KUKA KRL program: MyProgram_330().src

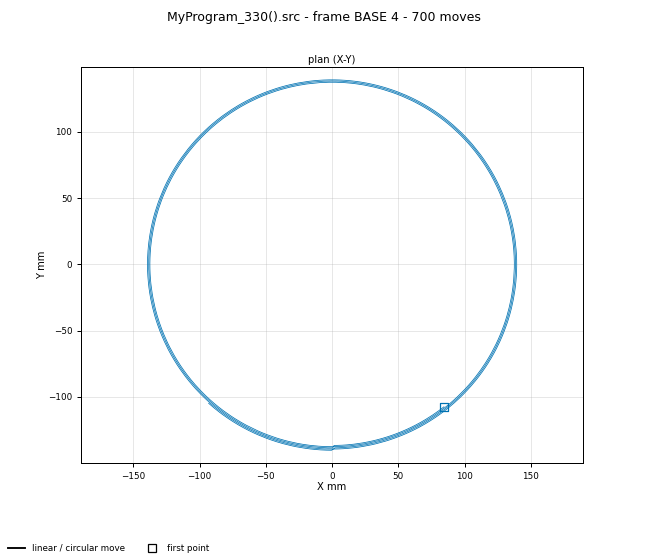
[picture p0: tool path of MyProgram_330().src in frame BASE 4, 700 of 700 moves have a stored position in this frame; points joined in program order, loops and branches not executed]
&ACCESS RVP
&REL 1
&PARAM TEMPLATE = C:\KRC\Roboter\Template\vorgabe
&PARAM EDITMASK = *
DEF MyProgram_330()
; ---- Setting reference (Base) ----
$BASE = BASE_DATA[4]

; --------------------------
; ---- Setting tool (TCP) ----
$TOOL = TOOL_DATA[3]
; --------------------------

$VEL.CP = VEL_APROX_PRINT
Startdeposition()
$VEL.CP = VEL_PRINT
LIN {X 84.385,Y -107.4322,Z 188,A -46.1092,B 2.2841,C 0.2483,E1 2.3985,E2 499.2761} C_DIS
LIN {X 80.7266,Y -110.2077,Z 188,A -48.0599,B 2.2837,C 0.2519,E1 2.3942,E2 501.2315} C_DIS
LIN {X 75.9214,Y -113.5713,Z 188,A -50.0705,B 2.2836,C 0.2529,E1 2.3897,E2 503.1841} C_DIS
LIN {X 73.4575,Y -115.1805,Z 188,A -51.7309,B 2.283,C 0.258,E1 2.3856,E2 504.9023} C_DIS
LIN {X 70.5993,Y -116.9539,Z 188,A -53.2982,B 2.2826,C 0.2614,E1 2.3818,E2 506.4914} C_DIS
LIN {X 66.6613,Y -119.2429,Z 188,A -54.7214,B 2.2826,C 0.2609,E1 2.3785,E2 507.8512} C_DIS
LIN {X 62.8545,Y -121.2922,Z 188,A -56.3872,B 2.2825,C 0.2626,E1 2.3744,E2 509.4986} C_DIS
LIN {X 59.8633,Y -122.7955,Z 188,A -57.8683,B 2.2822,C 0.2651,E1 2.3707,E2 510.991} C_DIS
LIN {X 56.2359,Y -124.4979,Z 188,A -59.8597,B 2.2817,C 0.2694,E1 2.3655,E2 513.0249} C_DIS
LIN {X 52.2998,Y -126.2016,Z 188,A -61.4901,B 2.2816,C 0.2705,E1 2.3614,E2 514.6342} C_DIS
LIN {X 48.8157,Y -127.5912,Z 188,A -62.7982,B 2.2816,C 0.2707,E1 2.358,E2 515.908} C_DIS
LIN {X 45.0187,Y -128.9782,Z 188,A -64.6024,B 2.2812,C 0.2733,E1 2.3532,E2 517.7279} C_DIS
LIN {X 41.9391,Y -130.0125,Z 188,A -65.4919,B 2.2814,C 0.2716,E1 2.351,E2 518.5549} C_DIS
LIN {X 37.8163,Y -131.2718,Z 188,A -67.5436,B 2.281,C 0.275,E1 2.3454,E2 520.6404} C_DIS
LIN {X 33.6424,Y -132.4016,Z 188,A -69.2051,B 2.281,C 0.2757,E1 2.341,E2 522.2827} C_DIS
LIN {X 30.2435,Y -133.2193,Z 188,A -70.6666,B 2.2808,C 0.2769,E1 2.337,E2 523.7444} C_DIS
LIN {X 26.7771,Y -133.9598,Z 188,A -72.0868,B 2.2808,C 0.2776,E1 2.3331,E2 525.1566} C_DIS
LIN {X 22.9551,Y -134.6675,Z 188,A -74.5642,B 2.2799,C 0.2839,E1 2.326,E2 527.7481} C_DIS
LIN {X 16.6479,Y -135.5918,Z 188,A -76.2129,B 2.2805,C 0.2793,E1 2.3218,E2 529.2614} C_DIS
LIN {X 10.9508,Y -136.1704,Z 188,A -78.8787,B 2.2802,C 0.282,E1 2.3143,E2 531.9641} C_DIS
LIN {X 7.4758,Y -136.4059,Z 188,A -80.9653,B 2.2797,C 0.2861,E1 2.3082,E2 534.1351} C_DIS
LIN {X 1.4605,Y -136.6033,Z 188,A -82.7052,B 2.2801,C 0.2824,E1 2.3036,E2 535.7715} C_DIS
LIN {X 1.4605,Y -136.6033,Z 188,A -82.7052,B 2.2801,C 0.2824,E1 2.3036,E2 535.7715} C_DIS
Enddeposition()
LIN {X 1.0092,Y -137.5035,Z 188,A -82.2384,B 2.2498,C 0.2786,E1 2.2744,E2 535.2539} C_DIS
Startdeposition()
$VEL.CP = VEL_PRINT
LIN {X 4.8877,Y -137.4225,Z 188,A -80.4582,B 2.25,C 0.2772,E1 2.2795,E2 533.4505} C_DIS
LIN {X 9.447,Y -137.1848,Z 188,A -78.1611,B 2.2504,C 0.2742,E1 2.2861,E2 531.0981} C_DIS
LIN {X 14.028,Y -136.7928,Z 188,A -76.6474,B 2.2502,C 0.2756,E1 2.2901,E2 529.6387} C_DIS
LIN {X 20.7914,Y -135.9277,Z 188,A -73.7592,B 2.2504,C 0.2736,E1 2.2982,E2 526.7425} C_DIS
LIN {X 24.9857,Y -135.2215,Z 188,A -71.9483,B 2.2506,C 0.2722,E1 2.3032,E2 524.9253} C_DIS
LIN {X 28.2124,Y -134.5853,Z 188,A -70.7396,B 2.2506,C 0.2722,E1 2.3064,E2 523.738} C_DIS
LIN {X 32.1471,Y -133.6978,Z 188,A -69.2265,B 2.2506,C 0.2718,E1 2.3105,E2 522.2468} C_DIS
LIN {X 35.1427,Y -132.9421,Z 188,A -67.9438,B 2.2508,C 0.2706,E1 2.3139,E2 520.9639} C_DIS
LIN {X 38.5637,Y -131.99,Z 188,A -66.5352,B 2.2508,C 0.2697,E1 2.3177,E2 519.564} C_DIS
LIN {X 41.3681,Y -131.139,Z 188,A -65.2923,B 2.2511,C 0.2683,E1 2.321,E2 518.3174} C_DIS
LIN {X 44.7036,Y -130.0393,Z 188,A -64.0619,B 2.2511,C 0.2683,E1 2.3242,E2 517.1178} C_DIS
LIN {X 47.8191,Y -128.9264,Z 188,A -62.5742,B 2.2513,C 0.2659,E1 2.3282,E2 515.6143} C_DIS
LIN {X 54.9877,Y -126.0358,Z 188,A -59.4365,B 2.2517,C 0.2625,E1 2.3363,E2 512.4858} C_DIS
LIN {X 58.7508,Y -124.3268,Z 188,A -57.6919,B 2.252,C 0.26,E1 2.3407,E2 510.737} C_DIS
LIN {X 62.1581,Y -122.6576,Z 188,A -56.2754,B 2.2522,C 0.2589,E1 2.3442,E2 509.3417} C_DIS
LIN {X 64.9016,Y -121.2305,Z 188,A -54.4156,B 2.2528,C 0.253,E1 2.349,E2 507.403} C_DIS
LIN {X 69.1543,Y -118.8562,Z 188,A -52.9164,B 2.2528,C 0.2536,E1 2.3525,E2 505.9749} C_DIS
LIN {X 72.9516,Y -116.5642,Z 188,A -51.1222,B 2.2531,C 0.251,E1 2.3567,E2 504.1867} C_DIS
LIN {X 77.4592,Y -113.6185,Z 188,A -48.9633,B 2.2534,C 0.2478,E1 2.3617,E2 502.0377} C_DIS
LIN {X 81.2164,Y -110.9639,Z 188,A -47.1203,B 2.2537,C 0.2449,E1 2.3659,E2 500.2032} C_DIS
LIN {X 84.798,Y -108.2513,Z 188,A -45.3204,B 2.254,C 0.242,E1 2.3699,E2 498.4117} C_DIS
LIN {X 88.2179,Y -105.483,Z 188,A -43.5989,B 2.2543,C 0.2394,E1 2.3735,E2 496.7039} C_DIS
LIN {X 91.488,Y -102.66,Z 188,A -41.8357,B 2.2547,C 0.2361,E1 2.3772,E2 494.9444} C_DIS
LIN {X 94.8941,Y -99.5196,Z 188,A -39.9954,B 2.255,C 0.2329,E1 2.381,E2 493.1147} C_DIS
LIN {X 98.0963,Y -96.3647,Z 188,A -38.3712,B 2.2552,C 0.2308,E1 2.3841,E2 491.5226} C_DIS
LIN {X 100.1859,Y -94.1905,Z 188,A -36.9746,B 2.2556,C 0.2271,E1 2.3868,E2 490.1062} C_DIS
LIN {X 103.1659,Y -90.9168,Z 188,A -35.2946,B 2.2559,C 0.2243,E1 2.3899,E2 488.447} C_DIS
LIN {X 105.9358,Y -87.6734,Z 188,A -33.5608,B 2.2562,C 0.2207,E1 2.393,E2 486.7176} C_DIS
LIN {X 108.3988,Y -84.6101,Z 188,A -31.9453,B 2.2566,C 0.2171,E1 2.3958,E2 485.1038} C_DIS
LIN {X 112.2568,Y -79.4196,Z 188,A -28.7306,B 2.2575,C 0.2067,E1 2.4012,E2 481.8167} C_DIS
LIN {X 115.783,Y -74.1843,Z 188,A -26.5211,B 2.2578,C 0.2037,E1 2.4045,E2 479.6621} C_DIS
LIN {X 118.237,Y -70.2074,Z 188,A -25.0755,B 2.2578,C 0.2029,E1 2.4064,E2 478.2823} C_DIS
LIN {X 120.3276,Y -66.5604,Z 188,A -23.5052,B 2.2582,C 0.2,E1 2.4086,E2 476.7348} C_DIS
LIN {X 122.3374,Y -62.7871,Z 188,A -21.8144,B 2.2585,C 0.1962,E1 2.4107,E2 475.0547} C_DIS
LIN {X 123.689,Y -60.0848,Z 188,A -20.6209,B 2.2587,C 0.1935,E1 2.4122,E2 473.869} C_DIS
LIN {X 125.4096,Y -56.4002,Z 188,A -19.1302,B 2.2589,C 0.1908,E1 2.4139,E2 472.404} C_DIS
LIN {X 127.1795,Y -52.2917,Z 188,A -17.2805,B 2.2593,C 0.186,E1 2.4159,E2 470.5549} C_DIS
LIN {X 128.6189,Y -48.64,Z 188,A -15.725,B 2.2596,C 0.1823,E1 2.4175,E2 469.0087} C_DIS
LIN {X 129.6006,Y -45.964,Z 188,A -14.34,B 2.26,C 0.1775,E1 2.4188,E2 467.5967} C_DIS
LIN {X 130.667,Y -42.8375,Z 188,A -13.3208,B 2.26,C 0.1768,E1 2.4197,E2 466.6238} C_DIS
LIN {X 131.8901,Y -38.905,Z 188,A -11.6877,B 2.2604,C 0.1728,E1 2.421,E2 465.0003} C_DIS
LIN {X 132.827,Y -35.5744,Z 188,A -10.3764,B 2.2606,C 0.17,E1 2.4219,E2 463.7052} C_DIS
LIN {X 133.5449,Y -32.7814,Z 188,A -9.1356,B 2.2609,C 0.1663,E1 2.4228,E2 462.4583} C_DIS
LIN {X 134.3884,Y -29.1259,Z 188,A -7.7687,B 2.2611,C 0.1637,E1 2.4236,E2 461.1161} C_DIS
LIN {X 135.0373,Y -25.9515,Z 188,A -6.4806,B 2.2613,C 0.1604,E1 2.4243,E2 459.8352} C_DIS
LIN {X 135.6371,Y -22.6082,Z 188,A -4.5754,B 2.2619,C 0.1524,E1 2.4252,E2 457.8646} C_DIS
LIN {X 136.364,Y -17.7048,Z 188,A -3.254,B 2.2619,C 0.1529,E1 2.4257,E2 456.6394} C_DIS
LIN {X 137.0505,Y -11.2195,Z 188,A -0.508,B 2.2623,C 0.145,E1 2.4264,E2 453.8881} C_DIS
LIN {X 137.4867,Y -2.4643,Z 188,A 3.1629,B 2.263,C 0.1346,E1 2.4268,E2 450.2126} C_DIS
LIN {X 137.5031,Y 1.4155,Z 188,A 4.4461,B 2.263,C 0.1328,E1 2.4268,E2 448.9718} C_DIS
LIN {X 137.3718,Y 6.1756,Z 188,A 6.7563,B 2.2636,C 0.1246,E1 2.4265,E2 446.6181} C_DIS
LIN {X 137.064,Y 11.0604,Z 188,A 8.1298,B 2.2636,C 0.1243,E1 2.4262,E2 445.3298} C_DIS
LIN {X 136.5849,Y 15.9147,Z 188,A 10.3416,B 2.264,C 0.1172,E1 2.4256,E2 443.0936} C_DIS
LIN {X 136.139,Y 19.3583,Z 188,A 11.2132,B 2.264,C 0.1179,E1 2.4253,E2 442.2952} C_DIS
LIN {X 135.4537,Y 23.6884,Z 188,A 13.1868,B 2.2642,C 0.1116,E1 2.4244,E2 440.3019} C_DIS
LIN {X 134.7483,Y 27.4126,Z 188,A 14.6147,B 2.2644,C 0.1085,E1 2.4236,E2 438.8925} C_DIS
LIN {X 133.981,Y 30.9474,Z 188,A 16.1028,B 2.2646,C 0.1045,E1 2.4227,E2 437.4062} C_DIS
LIN {X 132.9463,Y 35.1268,Z 188,A 17.7419,B 2.2647,C 0.1008,E1 2.4216,E2 435.786} C_DIS
LIN {X 132.0775,Y 38.2649,Z 188,A 18.8829,B 2.2648,C 0.0989,E1 2.4207,E2 434.6718} C_DIS
LIN {X 131.1193,Y 41.4299,Z 188,A 20.3392,B 2.265,C 0.0945,E1 2.4195,E2 433.2049} C_DIS
LIN {X 130.0245,Y 44.7462,Z 188,A 21.7058,B 2.2651,C 0.0913,E1 2.4183,E2 431.8489} C_DIS
LIN {X 126.6388,Y 53.5863,Z 188,A 25.2973,B 2.2654,C 0.0838,E1 2.4147,E2 428.3006} C_DIS
LIN {X 124.7724,Y 57.7956,Z 188,A 27.17,B 2.2656,C 0.0792,E1 2.4126,E2 426.4331} C_DIS
LIN {X 123.3269,Y 60.8189,Z 188,A 28.5186,B 2.2657,C 0.076,E1 2.4109,E2 425.09} C_DIS
LIN {X 121.8441,Y 63.7378,Z 188,A 29.7762,B 2.2657,C 0.0733,E1 2.4093,E2 423.8453} C_DIS
LIN {X 119.9629,Y 67.2158,Z 188,A 31.2497,B 2.2659,C 0.0706,E1 2.4074,E2 422.3931} C_DIS
LIN {X 118.3323,Y 70.0475,Z 188,A 32.7955,B 2.266,C 0.0658,E1 2.4051,E2 420.8239} C_DIS
LIN {X 115.9995,Y 73.8462,Z 188,A 34.3445,B 2.266,C 0.0636,E1 2.4029,E2 419.313} C_DIS
LIN {X 113.911,Y 77.028,Z 188,A 36.0298,B 2.2662,C 0.0591,E1 2.4003,E2 417.6148} C_DIS
LIN {X 111.2107,Y 80.878,Z 188,A 37.8786,B 2.2663,C 0.0553,E1 2.3973,E2 415.7793} C_DIS
LIN {X 108.5058,Y 84.4725,Z 188,A 39.6601,B 2.2663,C 0.0517,E1 2.3943,E2 414.0091} C_DIS
LIN {X 105.801,Y 87.8362,Z 188,A 41.375,B 2.2665,C 0.0483,E1 2.3913,E2 412.3041} C_DIS
LIN {X 102.8084,Y 91.3211,Z 188,A 43.0061,B 2.2665,C 0.0462,E1 2.3884,E2 410.7077} C_DIS
LIN {X 100.499,Y 93.8563,Z 188,A 44.5615,B 2.2665,C 0.0422,E1 2.3854,E2 409.1366} C_DIS
LIN {X 97.3828,Y 97.0858,Z 188,A 46.258,B 2.2666,C 0.0396,E1 2.3821,E2 407.4612} C_DIS
LIN {X 94.6427,Y 99.7593,Z 188,A 47.9247,B 2.2667,C 0.0358,E1 2.3787,E2 405.7856} C_DIS
LIN {X 90.7645,Y 103.3005,Z 188,A 49.998,B 2.2667,C 0.0323,E1 2.3744,E2 403.7263} C_DIS
LIN {X 87.3118,Y 106.2347,Z 188,A 51.8087,B 2.2667,C 0.0293,E1 2.3706,E2 401.9249} C_DIS
LIN {X 83.8262,Y 109.0061,Z 188,A 53.61,B 2.2668,C 0.0262,E1 2.3666,E2 400.1302} C_DIS
LIN {X 80.1135,Y 111.7625,Z 188,A 55.4244,B 2.2668,C 0.0236,E1 2.3625,E2 398.3296} C_DIS
LIN {X 76.6335,Y 114.1772,Z 188,A 56.9231,B 2.2668,C 0.0224,E1 2.3592,E2 396.8635} C_DIS
LIN {X 73.842,Y 116.0022,Z 188,A 58.4469,B 2.2669,C 0.0192,E1 2.3555,E2 395.3233} C_DIS
LIN {X 70.038,Y 118.338,Z 188,A 60.482,B 2.2669,C 0.0151,E1 2.3506,E2 393.267} C_DIS
LIN {X 67.0583,Y 120.0514,Z 188,A 61.6697,B 2.2669,C 0.0146,E1 2.3478,E2 392.1093} C_DIS
LIN {X 62.7474,Y 122.3576,Z 188,A 63.5951,B 2.2669,C 0.0123,E1 2.343,E2 390.1975} C_DIS
LIN {X 59.8978,Y 123.7788,Z 188,A 65.8423,B 2.2669,C 0.0047,E1 2.3371,E2 387.8377} C_DIS
LIN {X 53.1857,Y 126.8061,Z 188,A 67.5662,B 2.2669,C 0.0092,E1 2.3331,E2 386.2787} C_DIS
LIN {X 49.184,Y 128.4129,Z 188,A 69.6653,B 2.2669,C 0.0052,E1 2.3275,E2 384.1434} C_DIS
LIN {X 45.5722,Y 129.7381,Z 188,A 71.2409,B 2.2669,C 0.0036,E1 2.3234,E2 382.5715} C_DIS
LIN {X 41.6932,Y 131.0351,Z 188,A 72.7706,B 2.2669,C 0.0029,E1 2.3194,E2 381.0632} C_DIS
LIN {X 38.8098,Y 131.918,Z 188,A 73.9119,B 2.2669,C 0.0024,E1 2.3163,E2 379.9361} C_DIS
LIN {X 35.34,Y 132.8895,Z 188,A 75.5057,B 2.2669,C 0.0005,E1 2.312,E2 378.3315} C_DIS
LIN {X 31.2031,Y 133.9226,Z 188,A 77.3013,B 2.2669,C -0.0011,E1 2.3071,E2 376.5341} C_DIS
LIN {X 26.966,Y 134.8391,Z 188,A 79.1348,B 2.2669,C -0.0026,E1 2.3021,E2 374.6979} C_DIS
LIN {X 24,Y 135.3979,Z 188,A 80.9141,B 2.2669,C -0.0063,E1 2.297,E2 372.8556} C_DIS
LIN {X 18.5994,Y 136.2463,Z 188,A 82.5017,B 2.2669,C -0.0038,E1 2.2929,E2 371.3526} C_DIS
LIN {X 14.7664,Y 136.7133,Z 188,A 84.1663,B 2.2669,C -0.0049,E1 2.2882,E2 369.6818} C_DIS
LIN {X 9.7967,Y 137.1593,Z 188,A 86.1603,B 2.2669,C -0.0053,E1 2.2827,E2 367.6988} C_DIS
LIN {X 5.5957,Y 137.3949,Z 188,A 87.923,B 2.2669,C -0.0059,E1 2.2777,E2 365.9356} C_DIS
LIN {X 2.7166,Y 137.4825,Z 188,A 89.6743,B 2.2669,C -0.009,E1 2.2727,E2 364.1183} C_DIS
LIN {X -2.2082,Y 137.4909,Z 188,A 91.1797,B 2.2669,C -0.0066,E1 2.2686,E2 362.6798} C_DIS
LIN {X -9.3667,Y 137.1907,Z 188,A 94.2648,B 2.2669,C -0.0072,E1 2.26,E2 359.5841} C_DIS
LIN {X -19.2271,Y 136.1578,Z 188,A 98.2457,B 2.2669,C -0.0059,E1 2.249,E2 355.6234} C_DIS
LIN {X -22.1843,Y 135.7078,Z 188,A 99.3663,B 2.2669,C -0.005,E1 2.2459,E2 354.5186} C_DIS
LIN {X -25.6321,Y 135.0984,Z 188,A 100.9338,B 2.2669,C -0.005,E1 2.2416,E2 352.9388} C_DIS
LIN {X -28.9391,Y 134.4287,Z 188,A 102.2586,B 2.2669,C -0.0041,E1 2.2379,E2 351.6244} C_DIS
LIN {X -31.8422,Y 133.7713,Z 188,A 103.5303,B 2.2669,C -0.0037,E1 2.2345,E2 350.3497} C_DIS
LIN {X -35.1431,Y 132.942,Z 188,A 105.0418,B 2.2669,C -0.0033,E1 2.2303,E2 348.8277} C_DIS
LIN {X -37.9505,Y 132.1695,Z 188,A 106.3797,B 2.2669,C -0.0031,E1 2.2267,E2 347.4755} C_DIS
LIN {X -42.3548,Y 130.8238,Z 188,A 109.2577,B 2.2669,C -0.0056,E1 2.2188,E2 344.4824} C_DIS
LIN {X -49.02,Y 128.4766,Z 188,A 111.4022,B 2.2669,C -0.0001,E1 2.2134,E2 342.4369} C_DIS
LIN {X -51.732,Y 127.4064,Z 188,A 112.9877,B 2.2669,C -0.0004,E1 2.2092,E2 340.8072} C_DIS
LIN {X -55.7214,Y 125.7132,Z 188,A 114.397,B 2.2669,C 0.0028,E1 2.2057,E2 339.4471} C_DIS
LIN {X -59.0649,Y 124.1767,Z 188,A 115.8846,B 2.2669,C 0.0046,E1 2.2019,E2 337.9659} C_DIS
LIN {X -61.9449,Y 122.7661,Z 188,A 117.3342,B 2.2669,C 0.0056,E1 2.1982,E2 336.5036} C_DIS
LIN {X -64.7223,Y 121.3269,Z 188,A 118.7822,B 2.2669,C 0.0067,E1 2.1946,E2 335.039} C_DIS
LIN {X -68.9997,Y 118.9457,Z 188,A 120.7472,B 2.2669,C 0.0095,E1 2.1899,E2 333.0843} C_DIS
LIN {X -72.4713,Y 116.863,Z 188,A 122.6066,B 2.2669,C 0.0111,E1 2.1854,E2 331.2051} C_DIS
LIN {X -76.5464,Y 114.2354,Z 188,A 124.6275,B 2.2669,C 0.014,E1 2.1807,E2 329.1856} C_DIS
LIN {X -82.1038,Y 110.3086,Z 188,A 128.5193,B 2.2669,C 0.0151,E1 2.1716,E2 325.1665} C_DIS
LIN {X -87.6822,Y 105.9285,Z 188,A 131.1917,B 2.2669,C 0.0209,E1 2.1659,E2 322.531} C_DIS
LIN {X -91.5102,Y 102.64,Z 188,A 133.0073,B 2.2669,C 0.0254,E1 2.1622,E2 320.7521} C_DIS
LIN {X -95.4132,Y 99.0224,Z 188,A 135.1786,B 2.2668,C 0.0296,E1 2.1578,E2 318.5881} C_DIS
LIN {X -98.6463,Y 95.8017,Z 188,A 137.8599,B 2.2668,C 0.0311,E1 2.1524,E2 315.8122} C_DIS
LIN {X -102.6929,Y 91.4512,Z 188,A 139.5412,B 2.2667,C 0.0382,E1 2.1494,E2 314.2306} C_DIS
LIN {X -104.73,Y 89.1103,Z 188,A 141.5886,B 2.2667,C 0.0389,E1 2.1455,E2 312.0913} C_DIS
LIN {X -107.7808,Y 85.3956,Z 188,A 143.0983,B 2.2665,C 0.0444,E1 2.143,E2 310.6439} C_DIS
LIN {X -110.484,Y 81.8683,Z 188,A 145.1289,B 2.2665,C 0.048,E1 2.1395,E2 308.5927} C_DIS
LIN {X -112.9783,Y 78.3897,Z 188,A 146.9931,B 2.2664,C 0.0518,E1 2.1365,E2 306.7198} C_DIS
LIN {X -115.3932,Y 74.7893,Z 188,A 148.9146,B 2.2664,C 0.0557,E1 2.1335,E2 304.7854} C_DIS
LIN {X -117.1838,Y 71.9513,Z 188,A 150.7097,B 2.2662,C 0.0581,E1 2.1309,E2 302.9422} C_DIS
LIN {X -119.1363,Y 68.6704,Z 188,A 152.0071,B 2.2662,C 0.0625,E1 2.1291,E2 301.6824} C_DIS
LIN {X -121.3269,Y 64.7222,Z 188,A 154.1462,B 2.266,C 0.0665,E1 2.1262,E2 299.5126} C_DIS
LIN {X -123.331,Y 60.8105,Z 188,A 155.8989,B 2.2659,C 0.0712,E1 2.124,E2 297.771} C_DIS
LIN {X -124.5803,Y 58.211,Z 188,A 157.261,B 2.2658,C 0.0739,E1 2.1224,E2 296.3898} C_DIS
LIN {X -125.9787,Y 55.1199,Z 188,A 158.7316,B 2.2657,C 0.0774,E1 2.1207,E2 294.9131} C_DIS
LIN {X -127.2677,Y 52.0761,Z 188,A 160.275,B 2.2656,C 0.0806,E1 2.119,E2 293.35} C_DIS
LIN {X -128.6839,Y 48.4665,Z 188,A 161.8237,B 2.2654,C 0.0849,E1 2.1175,E2 291.8108} C_DIS
LIN {X -129.8655,Y 45.2048,Z 188,A 163.2663,B 2.2652,C 0.0887,E1 2.1161,E2 290.3696} C_DIS
LIN {X -130.721,Y 42.6749,Z 188,A 164.6068,B 2.2652,C 0.0912,E1 2.1149,E2 289.0014} C_DIS
LIN {X -131.9233,Y 38.7915,Z 188,A 166.4002,B 2.265,C 0.0955,E1 2.1135,E2 287.1967} C_DIS
LIN {X -133.2108,Y 34.1098,Z 188,A 168.5508,B 2.2647,C 0.1008,E1 2.1119,E2 285.0314} C_DIS
LIN {X -134.0307,Y 30.7299,Z 188,A 170.202,B 2.2646,C 0.1043,E1 2.1108,E2 283.3558} C_DIS
LIN {X -135.0028,Y 26.1323,Z 188,A 172.2053,B 2.2643,C 0.1096,E1 2.1097,E2 281.348} C_DIS
LIN {X -135.6278,Y 22.6641,Z 188,A 173.719,B 2.2641,C 0.1136,E1 2.109,E2 279.8296} C_DIS
LIN {X -136.0754,Y 19.8037,Z 188,A 175.0268,B 2.264,C 0.1167,E1 2.1084,E2 278.5098} C_DIS
LIN {X -136.4612,Y 16.9522,Z 188,A 176.4374,B 2.2638,C 0.1197,E1 2.1079,E2 277.073} C_DIS
LIN {X -136.9105,Y 12.8145,Z 188,A 178.2497,B 2.2636,C 0.1244,E1 2.1074,E2 275.252} C_DIS
LIN {X -137.2408,Y 8.5783,Z 188,A -179.9451,B 2.2633,C 0.1293,E1 2.1071,E2 273.4434} C_DIS
LIN {X -137.428,Y 4.7461,Z 188,A -178.274,B 2.263,C 0.1336,E1 2.1069,E2 271.7641} C_DIS
LIN {X -137.5082,Y 0.6532,Z 188,A -176.3294,B 2.2628,C 0.138,E1 2.1068,E2 269.7899} C_DIS
LIN {X -137.4625,Y -3.5713,Z 188,A -174.5103,B 2.2625,C 0.1428,E1 2.1068,E2 267.9644} C_DIS
LIN {X -137.3184,Y -7.2363,Z 188,A -172.8003,B 2.2622,C 0.1467,E1 2.1071,E2 266.2318} C_DIS
LIN {X -137.0681,Y -11.0116,Z 188,A -171.1578,B 2.262,C 0.151,E1 2.1075,E2 264.5817} C_DIS
LIN {X -136.6969,Y -14.9194,Z 188,A -169.4434,B 2.2617,C 0.1554,E1 2.108,E2 262.8581} C_DIS
LIN {X -136.1792,Y -19.0769,Z 188,A -167.5781,B 2.2613,C 0.16,E1 2.1086,E2 260.9783} C_DIS
LIN {X -135.7078,Y -22.1843,Z 188,A -166.274,B 2.2611,C 0.1636,E1 2.1092,E2 259.6756} C_DIS
LIN {X -135.1272,Y -25.4818,Z 188,A -164.6905,B 2.2608,C 0.1671,E1 2.11,E2 258.0683} C_DIS
LIN {X -134.4414,Y -28.8803,Z 188,A -163.2603,B 2.2605,C 0.1711,E1 2.1108,E2 256.6408} C_DIS
LIN {X -133.7519,Y -31.9227,Z 188,A -161.8533,B 2.2603,C 0.1744,E1 2.1117,E2 255.2205} C_DIS
LIN {X -133.0511,Y -34.7339,Z 188,A -160.4123,B 2.2601,C 0.1771,E1 2.1128,E2 253.7496} C_DIS
LIN {X -132.0466,Y -38.3704,Z 188,A -158.8371,B 2.2597,C 0.1813,E1 2.114,E2 252.1747} C_DIS
LIN {X -130.2796,Y -44.0009,Z 188,A -156.1023,B 2.2592,C 0.1872,E1 2.1163,E2 249.4049} C_DIS
LIN {X -128.555,Y -48.8107,Z 188,A -153.8695,B 2.2588,C 0.1925,E1 2.1185,E2 247.1593} C_DIS
LIN {X -126.9886,Y -52.7487,Z 188,A -152.0935,B 2.2584,C 0.197,E1 2.1204,E2 245.3827} C_DIS
LIN {X -125.5772,Y -56.0254,Z 188,A -150.6125,B 2.2581,C 0.2008,E1 2.122,E2 243.903} C_DIS
LIN {X -124.1951,Y -59.0265,Z 188,A -149.0837,B 2.2578,C 0.2039,E1 2.1239,E2 242.3546} C_DIS
LIN {X -122.6701,Y -62.1335,Z 188,A -147.5877,B 2.2575,C 0.2073,E1 2.1257,E2 240.8521} C_DIS
LIN {X -119.0182,Y -68.8745,Z 188,A -144.0569,B 2.2569,C 0.2141,E1 2.1306,E2 237.2779} C_DIS
LIN {X -116.6028,Y -72.8896,Z 188,A -141.9949,B 2.2564,C 0.2184,E1 2.1336,E2 235.2019} C_DIS
LIN {X -114.1602,Y -76.6591,Z 188,A -140.0279,B 2.2561,C 0.2223,E1 2.1366,E2 233.2228} C_DIS
LIN {X -111.6162,Y -80.3182,Z 188,A -138.0713,B 2.2557,C 0.2262,E1 2.1398,E2 231.2532} C_DIS
LIN {X -108.9478,Y -83.9022,Z 188,A -136.1116,B 2.2553,C 0.2299,E1 2.1431,E2 229.2809} C_DIS
LIN {X -106.2091,Y -87.3431,Z 188,A -134.1535,B 2.255,C 0.2333,E1 2.1466,E2 227.3063} C_DIS
LIN {X -103.5532,Y -90.4752,Z 188,A -131.6718,B 2.2548,C 0.2344,E1 2.1514,E2 224.7208} C_DIS
LIN {X -99.5157,Y -94.8982,Z 188,A -129.96,B 2.2541,C 0.2417,E1 2.1544,E2 223.1153} C_DIS
LIN {X -95.4652,Y -98.9721,Z 188,A -127.3581,B 2.2537,C 0.2455,E1 2.1597,E2 220.4857} C_DIS
LIN {X -92.369,Y -101.8675,Z 188,A -125.4795,B 2.2534,C 0.2482,E1 2.1636,E2 218.5922} C_DIS
LIN {X -88.9812,Y -104.8397,Z 188,A -123.4974,B 2.253,C 0.2511,E1 2.1678,E2 216.596} C_DIS
LIN {X -85.4608,Y -107.7289,Z 188,A -121.5416,B 2.2527,C 0.2539,E1 2.1721,E2 214.6324} C_DIS
LIN {X -81.8426,Y -110.5031,Z 188,A -119.549,B 2.2524,C 0.2565,E1 2.1765,E2 212.6273} C_DIS
LIN {X -79.3508,Y -112.3053,Z 188,A -118.042,B 2.2524,C 0.2576,E1 2.1801,E2 211.0896} C_DIS
LIN {X -76.6488,Y -114.167,Z 188,A -116.7829,B 2.252,C 0.2599,E1 2.1829,E2 209.8452} C_DIS
LIN {X -73.3109,Y -116.338,Z 188,A -114.9317,B 2.2519,C 0.2614,E1 2.1874,E2 207.9677} C_DIS
LIN {X -68.5317,Y -119.2166,Z 188,A -112.7023,B 2.2515,C 0.2647,E1 2.1927,E2 205.7512} C_DIS
LIN {X -64.629,Y -121.3762,Z 188,A -110.7882,B 2.2513,C 0.2666,E1 2.1974,E2 203.8293} C_DIS
LIN {X -56.1373,Y -125.5272,Z 188,A -107.0196,B 2.2507,C 0.2714,E1 2.2069,E2 200.0833} C_DIS
LIN {X -52.6904,Y -127.013,Z 188,A -105.2755,B 2.2507,C 0.272,E1 2.2114,E2 198.3144} C_DIS
LIN {X -48.9416,Y -128.5059,Z 188,A -103.3797,B 2.2506,C 0.2724,E1 2.2165,E2 196.3891} C_DIS
LIN {X -45.0592,Y -129.916,Z 188,A -101.8833,B 2.2503,C 0.2747,E1 2.2203,E2 194.9229} C_DIS
LIN {X -42.0191,Y -130.931,Z 188,A -100.5596,B 2.2502,C 0.2757,E1 2.2238,E2 193.6005} C_DIS
LIN {X -39.4366,Y -131.7344,Z 188,A -99.1642,B 2.2502,C 0.2751,E1 2.2277,E2 192.1682} C_DIS
LIN {X -35.8085,Y -132.7645,Z 188,A -97.6957,B 2.2501,C 0.2765,E1 2.2316,E2 190.7132} C_DIS
LIN {X -32.4912,Y -133.6149,Z 188,A -96.2887,B 2.25,C 0.2772,E1 2.2354,E2 189.3085} C_DIS
LIN {X -29.1508,Y -134.383,Z 188,A -94.8386,B 2.25,C 0.2777,E1 2.2394,E2 187.8549} C_DIS
LIN {X -26.43,Y -134.9459,Z 188,A -93.2028,B 2.2502,C 0.2757,E1 2.2441,E2 186.1531} C_DIS
LIN {X -22.2736,Y -135.6929,Z 188,A -91.9109,B 2.2498,C 0.2785,E1 2.2475,E2 184.9248} C_DIS
LIN {X -17.0251,Y -136.4523,Z 188,A -89.5947,B 2.2498,C 0.2783,E1 2.2539,E2 182.5932} C_DIS
LIN {X -13.3974,Y -136.8545,Z 188,A -88.2108,B 2.2498,C 0.2792,E1 2.2577,E2 181.2274} C_DIS
LIN {X -10.1008,Y -137.1371,Z 188,A -86.7431,B 2.2498,C 0.2787,E1 2.2619,E2 179.7468} C_DIS
LIN {X -5.8583,Y -137.3847,Z 188,A -85.1488,B 2.2497,C 0.2795,E1 2.2663,E2 178.176} C_DIS
LIN {X -2.4585,Y -137.4868,Z 188,A -83.3294,B 2.25,C 0.2771,E1 2.2715,E2 176.3007} C_DIS
LIN {X 1.0092,Y -137.5035,Z 188,A -82.2352,B 2.2498,C 0.2787,E1 2.2744,E2 175.254} C_DIS
Enddeposition()
LIN {X 1.0092,Y -137.5035,Z 188,A -82.2352,B 2.2498,C 0.2787,E1 2.2744,E2 175.254} C_DIS
Startdeposition()
$VEL.CP = VEL_PRINT
LIN {X 0.485,Y -138.4074,Z 188,A -82.9376,B 2.2195,C 0.2814,E1 2.2423,E2 176.0609} C_DIS
LIN {X -3.0721,Y -138.376,Z 188,A -84.3646,B 2.2195,C 0.2814,E1 2.2384,E2 177.4825} C_DIS
LIN {X -7.039,Y -138.2288,Z 188,A -86.0465,B 2.2195,C 0.2818,E1 2.2336,E2 179.1702} C_DIS
LIN {X -10.1831,Y -138.0328,Z 188,A -87.3397,B 2.2195,C 0.2818,E1 2.23,E2 180.4626} C_DIS
LIN {X -13.5165,Y -137.7466,Z 188,A -88.7025,B 2.2195,C 0.2816,E1 2.2262,E2 181.8229} C_DIS
LIN {X -16.6864,Y -137.3986,Z 188,A -90.0282,B 2.2195,C 0.2814,E1 2.2225,E2 183.1499} C_DIS
LIN {X -19.8727,Y -136.974,Z 188,A -91.3571,B 2.2195,C 0.2812,E1 2.2189,E2 184.4791} C_DIS
LIN {X -23.073,Y -136.4713,Z 188,A -92.7168,B 2.2195,C 0.281,E1 2.2151,E2 185.8419} C_DIS
LIN {X -26.7933,Y -135.792,Z 188,A -94.2952,B 2.2195,C 0.2806,E1 2.2107,E2 187.4227} C_DIS
LIN {X -29.5046,Y -135.2266,Z 188,A -95.5002,B 2.2195,C 0.2804,E1 2.2074,E2 188.636} C_DIS
LIN {X -33.2379,Y -134.3599,Z 188,A -97.0578,B 2.2197,C 0.2796,E1 2.2032,E2 190.1903} C_DIS
LIN {X -37.5738,Y -133.2102,Z 188,A -98.9409,B 2.2197,C 0.2787,E1 2.1981,E2 192.0773} C_DIS
LIN {X -40.8012,Y -132.2573,Z 188,A -100.3554,B 2.2199,C 0.278,E1 2.1943,E2 193.4951} C_DIS
LIN {X -44.5333,Y -131.0502,Z 188,A -102.0064,B 2.22,C 0.277,E1 2.1899,E2 195.1504} C_DIS
LIN {X -47.7465,Y -129.9139,Z 188,A -103.4434,B 2.2201,C 0.2761,E1 2.1861,E2 196.5913} C_DIS
LIN {X -50.948,Y -128.6921,Z 188,A -104.8906,B 2.2203,C 0.275,E1 2.1823,E2 198.0427} C_DIS
LIN {X -54.1346,Y -127.3845,Z 188,A -106.3474,B 2.2203,C 0.2739,E1 2.1785,E2 199.504} C_DIS
LIN {X -56.8432,Y -126.1966,Z 188,A -107.6427,B 2.2205,C 0.273,E1 2.1752,E2 200.8092} C_DIS
LIN {X -60.4494,Y -124.5119,Z 188,A -109.2885,B 2.2207,C 0.2714,E1 2.171,E2 202.455} C_DIS
LIN {X -63.571,Y -122.9475,Z 188,A -110.7721,B 2.2209,C 0.2699,E1 2.1673,E2 203.9439} C_DIS
LIN {X -67.1894,Y -121.0073,Z 188,A -112.5563,B 2.2211,C 0.2683,E1 2.1629,E2 205.7398} C_DIS
LIN {X -71.0034,Y -118.8095,Z 188,A -114.4332,B 2.2213,C 0.2663,E1 2.1584,E2 207.6243} C_DIS
LIN {X -74.6338,Y -116.5631,Z 188,A -116.284,B 2.2216,C 0.2642,E1 2.1539,E2 209.4866} C_DIS
LIN {X -78.1846,Y -114.2119,Z 188,A -118.1035,B 2.2218,C 0.262,E1 2.1497,E2 211.3137} C_DIS
LIN {X -81.586,Y -111.8082,Z 188,A -119.9338,B 2.2221,C 0.2598,E1 2.1455,E2 213.1585} C_DIS
LIN {X -85.2004,Y -109.0788,Z 188,A -121.8832,B 2.2224,C 0.2571,E1 2.1412,E2 215.1178} C_DIS
LIN {X -88.4021,Y -106.5,Z 188,A -123.5776,B 2.2227,C 0.2543,E1 2.1375,E2 216.8112} C_DIS
LIN {X -91.5867,Y -103.774,Z 188,A -125.4378,B 2.223,C 0.2518,E1 2.1335,E2 218.6881} C_DIS
LIN {X -94.8593,Y -100.7913,Z 188,A -127.3189,B 2.2234,C 0.2487,E1 2.1297,E2 220.5755} C_DIS
LIN {X -97.6696,Y -98.0705,Z 188,A -128.9762,B 2.2237,C 0.2458,E1 2.1263,E2 222.2378} C_DIS
LIN {X -100.6186,Y -95.0424,Z 188,A -130.8623,B 2.224,C 0.2429,E1 2.1227,E2 224.1419} C_DIS
LIN {X -103.5884,Y -91.7966,Z 188,A -132.7724,B 2.2244,C 0.2396,E1 2.1191,E2 226.0636} C_DIS
LIN {X -106.4846,Y -88.4207,Z 188,A -134.7097,B 2.2247,C 0.2361,E1 2.1155,E2 228.0134} C_DIS
LIN {X -109.1233,Y -85.1437,Z 188,A -136.442,B 2.2251,C 0.2324,E1 2.1125,E2 229.7442} C_DIS
LIN {X -111.4478,Y -82.0766,Z 188,A -138.2095,B 2.2254,C 0.2294,E1 2.1095,E2 231.5345} C_DIS
LIN {X -114.0868,Y -78.3668,Z 188,A -140.1818,B 2.2258,C 0.2255,E1 2.1064,E2 233.518} C_DIS
LIN {X -116.3311,Y -74.9962,Z 188,A -141.9385,B 2.2262,C 0.2219,E1 2.1037,E2 235.2849} C_DIS
LIN {X -118.6666,Y -71.2432,Z 188,A -143.8695,B 2.2266,C 0.2179,E1 2.1008,E2 237.2288} C_DIS
LIN {X -120.8727,Y -67.4326,Z 188,A -145.8558,B 2.227,C 0.214,E1 2.0981,E2 239.2361} C_DIS
LIN {X -122.8573,Y -63.7427,Z 188,A -147.5672,B 2.2274,C 0.2097,E1 2.0958,E2 240.9439} C_DIS
LIN {X -124.2678,Y -60.9444,Z 188,A -148.9571,B 2.2276,C 0.2068,E1 2.0941,E2 242.3455} C_DIS
LIN {X -125.991,Y -57.3028,Z 188,A -150.7003,B 2.228,C 0.2028,E1 2.092,E2 244.0981} C_DIS
LIN {X -127.1674,Y -54.6367,Z 188,A -151.9791,B 2.2283,C 0.1999,E1 2.0906,E2 245.3859} C_DIS
LIN {X -128.6167,Y -51.135,Z 188,A -153.6523,B 2.2286,C 0.1961,E1 2.0888,E2 247.0722} C_DIS
LIN {X -129.724,Y -48.2536,Z 188,A -155.0005,B 2.2289,C 0.1929,E1 2.0875,E2 248.429} C_DIS
LIN {X -130.8524,Y -45.1037,Z 188,A -156.4808,B 2.2292,C 0.1895,E1 2.0861,E2 249.9212} C_DIS
LIN {X -132.1011,Y -41.3116,Z 188,A -158.2293,B 2.2295,C 0.1854,E1 2.0846,E2 251.6816} C_DIS
LIN {X -132.9138,Y -38.609,Z 188,A -159.4637,B 2.2298,C 0.1824,E1 2.0836,E2 252.9239} C_DIS
LIN {X -133.8131,Y -35.3666,Z 188,A -160.9369,B 2.2301,C 0.1788,E1 2.0825,E2 254.407} C_DIS
LIN {X -134.625,Y -32.1384,Z 188,A -162.4204,B 2.2303,C 0.1753,E1 2.0815,E2 255.9035} C_DIS
LIN {X -135.3386,Y -28.9861,Z 188,A -163.8558,B 2.2306,C 0.1718,E1 2.0806,E2 257.3509} C_DIS
LIN {X -136.0021,Y -25.6943,Z 188,A -165.3754,B 2.2309,C 0.1683,E1 2.0798,E2 258.8866} C_DIS
LIN {X -136.6541,Y -21.9775,Z 188,A -166.9914,B 2.2312,C 0.1641,E1 2.0791,E2 260.5088} C_DIS
LIN {X -137.2428,Y -17.9205,Z 188,A -168.8288,B 2.2315,C 0.1596,E1 2.0783,E2 262.3633} C_DIS
LIN {X -137.6986,Y -14.0163,Z 188,A -170.5358,B 2.2318,C 0.1553,E1 2.0778,E2 264.0797} C_DIS
LIN {X -137.9832,Y -10.8621,Z 188,A -171.9337,B 2.2321,C 0.1518,E1 2.0775,E2 265.4881} C_DIS
LIN {X -138.2477,Y -6.6635,Z 188,A -173.7907,B 2.2324,C 0.1471,E1 2.0772,E2 267.3588} C_DIS
LIN {X -138.3624,Y -3.5614,Z 188,A -175.1613,B 2.2326,C 0.1437,E1 2.0771,E2 268.7396} C_DIS
LIN {X -138.4113,Y 0,Z 188,A -176.7772,B 2.2328,C 0.1398,E1 2.0771,E2 270.3728} C_DIS
LIN {X -138.376,Y 3.0721,Z 188,A -178.098,B 2.2331,C 0.1363,E1 2.0771,E2 271.699} C_DIS
LIN {X -138.2725,Y 6.1704,Z 188,A -179.4725,B 2.2333,C 0.1329,E1 2.0772,E2 273.0843} C_DIS
LIN {X -138.0363,Y 10.1358,Z 188,A 178.7293,B 2.2335,C 0.1285,E1 2.0776,E2 274.901} C_DIS
LIN {X -137.7466,Y 13.5165,Z 188,A 177.2625,B 2.2337,C 0.1247,E1 2.0779,E2 276.3747} C_DIS
LIN {X -137.3986,Y 16.6864,Z 188,A 175.8496,B 2.2339,C 0.1212,E1 2.0784,E2 277.7986} C_DIS
LIN {X -136.974,Y 19.8727,Z 188,A 174.4257,B 2.2341,C 0.1177,E1 2.079,E2 279.2334} C_DIS
LIN {X -136.4713,Y 23.073,Z 188,A 172.9913,B 2.2343,C 0.1141,E1 2.0796,E2 280.6787} C_DIS
LIN {X -135.873,Y 26.37,Z 188,A 171.4729,B 2.2345,C 0.1106,E1 2.0804,E2 282.2128} C_DIS
LIN {X -135.2266,Y 29.5046,Z 188,A 170.0424,B 2.2347,C 0.1071,E1 2.0812,E2 283.6556} C_DIS
LIN {X -134.3591,Y 33.2412,Z 188,A 168.3961,B 2.2348,C 0.1029,E1 2.0823,E2 285.3083} C_DIS
LIN {X -133.5188,Y 36.4702,Z 188,A 166.9214,B 2.235,C 0.0994,E1 2.0834,E2 286.7937} C_DIS
LIN {X -132.7443,Y 39.1879,Z 188,A 165.6724,B 2.2351,C 0.0964,E1 2.0844,E2 288.0517} C_DIS
LIN {X -131.7492,Y 42.4133,Z 188,A 164.1315,B 2.2353,C 0.0929,E1 2.0857,E2 289.6096} C_DIS
LIN {X -130.4927,Y 46.1411,Z 188,A 162.447,B 2.2355,C 0.0887,E1 2.0872,E2 291.3} C_DIS
LIN {X -129.4749,Y 48.9187,Z 188,A 161.1202,B 2.2355,C 0.0857,E1 2.0885,E2 292.6386} C_DIS
LIN {X -128.049,Y 52.5434,Z 188,A 159.4265,B 2.2357,C 0.0817,E1 2.0903,E2 294.3413} C_DIS
LIN {X -126.6985,Y 55.7212,Z 188,A 157.9066,B 2.2358,C 0.0782,E1 2.092,E2 295.8714} C_DIS
LIN {X -125.2622,Y 58.8791,Z 188,A 156.3807,B 2.236,C 0.0748,E1 2.0938,E2 297.4073} C_DIS
LIN {X -123.9242,Y 61.6408,Z 188,A 155.0004,B 2.236,C 0.0719,E1 2.0955,E2 298.8003} C_DIS
LIN {X -122.1334,Y 65.1213,Z 188,A 153.3138,B 2.2362,C 0.068,E1 2.0977,E2 300.494} C_DIS
LIN {X -120.1439,Y 68.7215,Z 188,A 151.471,B 2.2362,C 0.0642,E1 2.1002,E2 302.3527} C_DIS
LIN {X -118.0636,Y 72.2369,Z 188,A 149.6523,B 2.2364,C 0.0605,E1 2.1029,E2 304.1859} C_DIS
LIN {X -115.7906,Y 75.8276,Z 188,A 147.7558,B 2.2364,C 0.0568,E1 2.1058,E2 306.0979} C_DIS
LIN {X -113.5213,Y 79.1839,Z 188,A 146.0916,B 2.2366,C 0.0529,E1 2.1084,E2 307.7594} C_DIS
LIN {X -111.4478,Y 82.0766,Z 188,A 144.4998,B 2.2366,C 0.05,E1 2.111,E2 309.3645} C_DIS
LIN {X -108.8062,Y 85.5474,Z 188,A 142.6216,B 2.2367,C 0.0462,E1 2.1142,E2 311.2504} C_DIS
LIN {X -106.5,Y 88.4021,Z 188,A 141.0415,B 2.2367,C 0.0432,E1 2.117,E2 312.8367} C_DIS
LIN {X -104.1798,Y 91.125,Z 188,A 139.4873,B 2.2369,C 0.0403,E1 2.1199,E2 314.3988} C_DIS
LIN {X -101.5961,Y 93.9978,Z 188,A 137.7395,B 2.2369,C 0.0375,E1 2.1232,E2 316.1635} C_DIS
LIN {X -98.5972,Y 97.1383,Z 188,A 135.8423,B 2.2369,C 0.0343,E1 2.1269,E2 318.0714} C_DIS
LIN {X -95.5096,Y 100.1754,Z 188,A 134.0569,B 2.237,C 0.031,E1 2.1305,E2 319.8547} C_DIS
LIN {X -92.6756,Y 102.8037,Z 188,A 132.3881,B 2.237,C 0.0283,E1 2.134,E2 321.5307} C_DIS
LIN {X -89.7707,Y 105.349,Z 188,A 130.6403,B 2.237,C 0.0259,E1 2.1377,E2 323.2954} C_DIS
LIN {X -86.3232,Y 108.1919,Z 188,A 128.7378,B 2.237,C 0.023,E1 2.1418,E2 325.2029} C_DIS
LIN {X -83.2437,Y 110.5788,Z 188,A 127.0894,B 2.2371,C 0.0206,E1 2.1455,E2 326.8545} C_DIS
LIN {X -80.1414,Y 112.8482,Z 188,A 125.4795,B 2.2371,C 0.0182,E1 2.1492,E2 328.4656} C_DIS
LIN {X -76.9559,Y 115.0433,Z 188,A 123.7289,B 2.2371,C 0.0163,E1 2.1533,E2 330.233} C_DIS
LIN {X -73.2648,Y 117.4285,Z 188,A 121.8446,B 2.2371,C 0.0141,E1 2.1577,E2 332.1239} C_DIS
LIN {X -69.4843,Y 119.7043,Z 188,A 119.9638,B 2.2371,C 0.0119,E1 2.1623,E2 334.01} C_DIS
LIN {X -65.3658,Y 122.0021,Z 188,A 118.0213,B 2.2371,C 0.0095,E1 2.167,E2 335.95} C_DIS
LIN {X -62.0136,Y 123.7403,Z 188,A 116.4551,B 2.2372,C 0.0077,E1 2.1709,E2 337.5156} C_DIS
LIN {X -59.3351,Y 125.0443,Z 188,A 115.1492,B 2.2372,C 0.0067,E1 2.1743,E2 338.8294} C_DIS
LIN {X -55.7212,Y 126.6985,Z 188,A 113.5102,B 2.2372,C 0.005,E1 2.1784,E2 340.4667} C_DIS
LIN {X -53.0469,Y 127.8387,Z 188,A 112.2768,B 2.2372,C 0.004,E1 2.1816,E2 341.7029} C_DIS
LIN {X -49.7256,Y 129.1673,Z 188,A 110.7863,B 2.2372,C 0.0028,E1 2.1855,E2 343.1936} C_DIS
LIN {X -46.6492,Y 130.3096,Z 188,A 109.3909,B 2.2372,C 0.0018,E1 2.1892,E2 344.5927} C_DIS
LIN {X -43.4328,Y 131.4166,Z 188,A 107.9582,B 2.2372,C 0.0009,E1 2.193,E2 346.0275} C_DIS
LIN {X -40.0173,Y 132.4972,Z 188,A 106.436,B 2.2372,C 0,E1 2.1971,E2 347.5536} C_DIS
LIN {X -36.4702,Y 133.5188,Z 188,A 104.9095,B 2.2372,C -0.0009,E1 2.2012,E2 349.0791} C_DIS
LIN {X -33.7521,Y 134.2295,Z 188,A 103.7347,B 2.2372,C -0.0014,E1 2.2044,E2 350.2546} C_DIS
LIN {X -30.525,Y 135,Z 188,A 102.3058,B 2.2372,C -0.0018,E1 2.2083,E2 351.6894} C_DIS
LIN {X -27.4329,Y 135.6619,Z 188,A 101.0117,B 2.2372,C -0.0024,E1 2.2118,E2 352.9811} C_DIS
LIN {X -23.5801,Y 136.3867,Z 188,A 99.397,B 2.2372,C -0.0029,E1 2.2163,E2 354.594} C_DIS
LIN {X -20.3778,Y 136.9018,Z 188,A 98.0491,B 2.2372,C -0.0033,E1 2.22,E2 355.9419} C_DIS
LIN {X -17.1891,Y 137.3386,Z 188,A 96.7132,B 2.2372,C -0.0035,E1 2.2237,E2 357.2775} C_DIS
LIN {X -13.5165,Y 137.7466,Z 188,A 95.1406,B 2.2372,C -0.0035,E1 2.2281,E2 358.8545} C_DIS
LIN {X -10.0196,Y 138.0447,Z 188,A 93.697,B 2.2372,C -0.0035,E1 2.2321,E2 360.2963} C_DIS
LIN {X -6.6635,Y 138.2477,Z 188,A 92.3432,B 2.2372,C -0.0037,E1 2.2359,E2 361.645} C_DIS
LIN {X -3.5614,Y 138.3624,Z 188,A 91.0635,B 2.2372,C -0.0037,E1 2.2395,E2 362.9234} C_DIS
LIN {X -0.485,Y 138.4074,Z 188,A 89.7527,B 2.2372,C -0.0032,E1 2.2431,E2 364.2382} C_DIS
LIN {X 3.9735,Y 138.351,Z 188,A 87.9501,B 2.2372,C -0.003,E1 2.2482,E2 366.0349} C_DIS
LIN {X 7.7286,Y 138.1941,Z 188,A 86.4087,B 2.2372,C -0.0026,E1 2.2525,E2 367.574} C_DIS
LIN {X 11.9384,Y 137.8923,Z 188,A 84.6731,B 2.2372,C -0.002,E1 2.2573,E2 369.3075} C_DIS
LIN {X 15.0992,Y 137.582,Z 188,A 83.3702,B 2.2372,C -0.0014,E1 2.2609,E2 370.6086} C_DIS
LIN {X 18.1043,Y 137.2187,Z 188,A 82.1052,B 2.2372,C -0.0007,E1 2.2645,E2 371.8746} C_DIS
LIN {X 21.4435,Y 136.7368,Z 188,A 80.7461,B 2.2372,C 0,E1 2.2682,E2 373.2287} C_DIS
LIN {X 24.6775,Y 136.1903,Z 188,A 79.3646,B 2.2372,C 0.001,E1 2.272,E2 374.6126} C_DIS
LIN {X 28.4031,Y 135.4645,Z 188,A 77.8621,B 2.2372,C 0.0018,E1 2.2761,E2 376.1066} C_DIS
LIN {X 31.0748,Y 134.8744,Z 188,A 76.7379,B 2.2372,C 0.0026,E1 2.2792,E2 377.2294} C_DIS
LIN {X 34.4263,Y 134.0584,Z 188,A 75.3109,B 2.2372,C 0.0038,E1 2.2831,E2 378.6559} C_DIS
LIN {X 37.5738,Y 133.2102,Z 188,A 74.0208,B 2.2372,C 0.0047,E1 2.2865,E2 379.9385} C_DIS
LIN {X 40.8012,Y 132.2573,Z 188,A 72.6561,B 2.2372,C 0.0059,E1 2.2902,E2 381.2995} C_DIS
LIN {X 44.5333,Y 131.0502,Z 188,A 71.0683,B 2.2372,C 0.0074,E1 2.2944,E2 382.8828} C_DIS
LIN {X 47.7465,Y 129.9139,Z 188,A 69.6906,B 2.2372,C 0.0088,E1 2.298,E2 384.2561} C_DIS
LIN {X 50.442,Y 128.8888,Z 188,A 68.5286,B 2.2372,C 0.01,E1 2.301,E2 385.414} C_DIS
LIN {X 53.7156,Y 127.5595,Z 188,A 67.0677,B 2.2372,C 0.0117,E1 2.3048,E2 386.8746} C_DIS
LIN {X 57.3028,Y 125.991,Z 188,A 65.5259,B 2.2372,C 0.0134,E1 2.3087,E2 388.4067} C_DIS
LIN {X 60.4494,Y 124.5119,Z 188,A 64.1282,B 2.2372,C 0.015,E1 2.3122,E2 389.7992} C_DIS
LIN {X 63.2719,Y 123.0997,Z 188,A 62.775,B 2.2372,C 0.0172,E1 2.3156,E2 391.1577} C_DIS
LIN {X 67.4326,Y 120.8727,Z 188,A 60.8713,B 2.2372,C 0.0198,E1 2.3203,E2 393.0553} C_DIS
LIN {X 71.2115,Y 118.6855,Z 188,A 59.1542,B 2.2372,C 0.022,E1 2.3244,E2 394.7615} C_DIS
LIN {X 74.9962,Y 116.3311,Z 188,A 57.4421,B 2.2371,C 0.0241,E1 2.3284,E2 396.4574} C_DIS
LIN {X 78.1404,Y 114.2422,Z 188,A 55.8674,B 2.2371,C 0.0268,E1 2.332,E2 398.0334} C_DIS
LIN {X 81.586,Y 111.8082,Z 188,A 54.2559,B 2.2371,C 0.029,E1 2.3357,E2 399.6286} C_DIS
LIN {X 84.6617,Y 109.497,Z 188,A 52.6679,B 2.237,C 0.0319,E1 2.3392,E2 401.216} C_DIS
LIN {X 87.7126,Y 107.0686,Z 188,A 51.1154,B 2.237,C 0.0345,E1 2.3426,E2 402.7611} C_DIS
LIN {X 91.125,Y 104.1798,Z 188,A 49.4031,B 2.237,C 0.0371,E1 2.3462,E2 404.4565} C_DIS
LIN {X 93.9978,Y 101.5961,Z 188,A 47.8724,B 2.2369,C 0.0398,E1 2.3493,E2 405.979} C_DIS
LIN {X 96.9292,Y 98.8023,Z 188,A 46.2031,B 2.2369,C 0.0431,E1 2.3527,E2 407.6476} C_DIS
LIN {X 100.1754,Y 95.5096,Z 188,A 44.443,B 2.2367,C 0.046,E1 2.3561,E2 409.389} C_DIS
LIN {X 102.8037,Y 92.6756,Z 188,A 42.8317,B 2.2367,C 0.0496,E1 2.3591,E2 411.002} C_DIS
LIN {X 105.7449,Y 89.3049,Z 188,A 41.154,B 2.2367,C 0.0524,E1 2.3621,E2 412.6586} C_DIS
LIN {X 108.0159,Y 86.5443,Z 188,A 39.7464,B 2.2365,C 0.0552,E1 2.3646,E2 414.0576} C_DIS
LIN {X 110.4162,Y 83.4592,Z 188,A 38.1267,B 2.2365,C 0.0589,E1 2.3673,E2 415.6777} C_DIS
LIN {X 113.0104,Y 79.9115,Z 188,A 36.4248,B 2.2364,C 0.0623,E1 2.3701,E2 417.3655} C_DIS
LIN {X 115.3611,Y 76.4799,Z 188,A 34.8485,B 2.2363,C 0.0653,E1 2.3725,E2 418.9242} C_DIS
LIN {X 117.4035,Y 73.305,Z 188,A 33.2887,B 2.2362,C 0.069,E1 2.3749,E2 420.4841} C_DIS
LIN {X 119.7043,Y 69.4843,Z 188,A 31.5285,B 2.236,C 0.0729,E1 2.3774,E2 422.2341} C_DIS
LIN {X 121.9708,Y 65.424,Z 188,A 29.7743,B 2.236,C 0.0764,E1 2.3797,E2 423.9676} C_DIS
LIN {X 123.7403,Y 62.0136,Z 188,A 28.2968,B 2.2358,C 0.0796,E1 2.3815,E2 425.4315} C_DIS
LIN {X 125.2622,Y 58.8791,Z 188,A 26.9347,B 2.2357,C 0.0827,E1 2.3832,E2 426.7841} C_DIS
LIN {X 126.6884,Y 55.7438,Z 188,A 25.5924,B 2.2356,C 0.0857,E1 2.3847,E2 428.1165} C_DIS
LIN {X 128.049,Y 52.5434,Z 188,A 24.2315,B 2.2355,C 0.0889,E1 2.3862,E2 429.468} C_DIS
LIN {X 129.3137,Y 49.3489,Z 188,A 22.8909,B 2.2353,C 0.092,E1 2.3875,E2 430.7989} C_DIS
LIN {X 130.3096,Y 46.6492,Z 188,A 21.7689,B 2.2353,C 0.0946,E1 2.3886,E2 431.9126} C_DIS
LIN {X 131.4166,Y 43.4328,Z 188,A 20.4293,B 2.2351,C 0.0978,E1 2.3898,E2 433.2442} C_DIS
LIN {X 132.5948,Y 39.6986,Z 188,A 18.9165,B 2.2349,C 0.1014,E1 2.391,E2 434.744} C_DIS
LIN {X 133.5188,Y 36.4702,Z 188,A 17.6086,B 2.2348,C 0.1045,E1 2.392,E2 436.0422} C_DIS
LIN {X 134.2267,Y 33.7629,Z 188,A 16.5283,B 2.2347,C 0.107,E1 2.3927,E2 437.113} C_DIS
LIN {X 135,Y 30.525,Z 188,A 15.1807,B 2.2345,C 0.1105,E1 2.3936,E2 438.4575} C_DIS
LIN {X 135.6884,Y 27.3027,Z 188,A 13.9419,B 2.2343,C 0.1133,E1 2.3943,E2 439.681} C_DIS
LIN {X 136.3867,Y 23.5801,Z 188,A 12.4682,B 2.2342,C 0.1169,E1 2.395,E2 441.1436} C_DIS
LIN {X 136.9018,Y 20.3778,Z 188,A 11.207,B 2.234,C 0.12,E1 2.3955,E2 442.3951} C_DIS
LIN {X 137.3386,Y 17.1891,Z 188,A 9.9555,B 2.2338,C 0.123,E1 2.396,E2 443.6369} C_DIS
LIN {X 137.6986,Y 14.0163,Z 188,A 8.7143,B 2.2337,C 0.1261,E1 2.3963,E2 444.8685} C_DIS
LIN {X 137.9832,Y 10.8621,Z 188,A 7.4837,B 2.2335,C 0.1291,E1 2.3966,E2 446.0895} C_DIS
LIN {X 138.2404,Y 6.8095,Z 188,A 5.8892,B 2.2333,C 0.1331,E1 2.3969,E2 447.6739} C_DIS
LIN {X 138.3624,Y 3.5614,Z 188,A 4.6433,B 2.2331,C 0.136,E1 2.3969,E2 448.9077} C_DIS
LIN {X 138.4113,Y 0,Z 188,A 3.2221,B 2.2328,C 0.1398,E1 2.397,E2 450.323} C_DIS
LIN {X 138.376,Y -3.0721,Z 188,A 2.0594,B 2.2327,C 0.1424,E1 2.397,E2 451.4724} C_DIS
LIN {X 138.2477,Y -6.6635,Z 188,A 0.611,B 2.2324,C 0.1463,E1 2.3968,E2 452.9166} C_DIS
LIN {X 138.0365,Y -10.1329,Z 188,A -0.7311,B 2.2322,C 0.1495,E1 2.3966,E2 454.2471} C_DIS
LIN {X 137.7466,Y -13.5165,Z 188,A -2.0235,B 2.232,C 0.1525,E1 2.3962,E2 455.5256} C_DIS
LIN {X 137.4044,Y -16.6379,Z 188,A -3.2541,B 2.2318,C 0.1556,E1 2.3958,E2 456.7481} C_DIS
LIN {X 136.974,Y -19.8727,Z 188,A -4.5217,B 2.2316,C 0.1587,E1 2.3954,E2 458.0058} C_DIS
LIN {X 136.4713,Y -23.073,Z 188,A -5.7857,B 2.2314,C 0.1618,E1 2.3948,E2 459.2606} C_DIS
LIN {X 135.792,Y -26.7933,Z 188,A -7.2609,B 2.2311,C 0.1654,E1 2.394,E2 460.7252} C_DIS
LIN {X 135.2266,Y -29.5046,Z 188,A -8.3855,B 2.2309,C 0.1684,E1 2.3934,E2 461.8477} C_DIS
LIN {X 134.3591,Y -33.2412,Z 188,A -9.8398,B 2.2306,C 0.1716,E1 2.3924,E2 463.2857} C_DIS
LIN {X 133.5188,Y -36.4702,Z 188,A -11.1427,B 2.2304,C 0.1748,E1 2.3915,E2 464.5793} C_DIS
LIN {X 132.7443,Y -39.1879,Z 188,A -12.247,B 2.2302,C 0.1774,E1 2.3907,E2 465.6758} C_DIS
LIN {X 131.7492,Y -42.4133,Z 188,A -13.6098,B 2.2299,C 0.1809,E1 2.3895,E2 467.035} C_DIS
LIN {X 130.4927,Y -46.1411,Z 188,A -15.103,B 2.2296,C 0.1842,E1 2.3882,E2 468.5116} C_DIS
LIN {X 129.5074,Y -48.8319,Z 188,A -16.2332,B 2.2294,C 0.1869,E1 2.3871,E2 469.6352} C_DIS
LIN {X 128.049,Y -52.5434,Z 188,A -17.7834,B 2.2291,C 0.1904,E1 2.3855,E2 471.1735} C_DIS
LIN {X 126.7377,Y -55.6305,Z 188,A -19.0978,B 2.2288,C 0.1934,E1 2.384,E2 472.4792} C_DIS
LIN {X 125.2622,Y -58.8791,Z 188,A -20.4929,B 2.2286,C 0.1966,E1 2.3824,E2 473.8645} C_DIS
LIN {X 123.8486,Y -61.7941,Z 188,A -21.7724,B 2.2283,C 0.1996,E1 2.3808,E2 475.1369} C_DIS
LIN {X 122.1334,Y -65.1213,Z 188,A -23.3442,B 2.2279,C 0.2037,E1 2.3788,E2 476.7129} C_DIS
LIN {X 120.0059,Y -68.9633,Z 188,A -25.0672,B 2.2276,C 0.2074,E1 2.3764,E2 478.4247} C_DIS
LIN {X 117.7478,Y -72.7517,Z 188,A -26.7637,B 2.2273,C 0.2109,E1 2.374,E2 480.1053} C_DIS
LIN {X 115.3611,Y -76.4799,Z 188,A -28.4838,B 2.2269,C 0.2144,E1 2.3714,E2 481.812} C_DIS
LIN {X 113.0104,Y -79.9115,Z 188,A -30.0905,B 2.2266,C 0.2176,E1 2.3689,E2 483.4046} C_DIS
LIN {X 110.7488,Y -83.0185,Z 188,A -31.5682,B 2.2263,C 0.2205,E1 2.3664,E2 484.8684} C_DIS
LIN {X 108.572,Y -85.8457,Z 188,A -33.0852,B 2.226,C 0.2241,E1 2.3638,E2 486.3919} C_DIS
LIN {X 105.6903,Y -89.3691,Z 188,A -34.866,B 2.2256,C 0.2276,E1 2.3607,E2 488.1603} C_DIS
LIN {X 102.9926,Y -92.4646,Z 188,A -36.4213,B 2.2253,C 0.2302,E1 2.3578,E2 489.6976} C_DIS
LIN {X 100.3712,Y -95.3046,Z 188,A -37.9787,B 2.225,C 0.2333,E1 2.3548,E2 491.2505} C_DIS
LIN {X 97.3448,Y -98.3933,Z 188,A -39.6862,B 2.2247,C 0.2364,E1 2.3515,E2 492.9483} C_DIS
LIN {X 94.2052,Y -101.403,Z 188,A -41.378,B 2.2244,C 0.2393,E1 2.3481,E2 494.6268} C_DIS
LIN {X 91.3383,Y -103.9936,Z 188,A -42.874,B 2.2241,C 0.2417,E1 2.345,E2 496.1102} C_DIS
LIN {X 88.4231,Y -106.4827,Z 188,A -44.4827,B 2.2238,C 0.2449,E1 2.3415,E2 497.7229} C_DIS
LIN {X 84.9358,Y -109.2845,Z 188,A -46.2314,B 2.2235,C 0.2476,E1 2.3377,E2 499.4592} C_DIS
LIN {X 81.586,Y -111.8082,Z 188,A -47.8379,B 2.2232,C 0.2498,E1 2.3342,E2 501.0495} C_DIS
LIN {X 78.6852,Y -113.8683,Z 188,A -49.3175,B 2.2229,C 0.2524,E1 2.3308,E2 502.5311} C_DIS
LIN {X 75.1241,Y -116.2481,Z 188,A -51.041,B 2.2226,C 0.2551,E1 2.3268,E2 504.2492} C_DIS
LIN {X 71.2432,Y -118.6666,Z 188,A -52.8491,B 2.2224,C 0.2575,E1 2.3225,E2 506.0472} C_DIS
LIN {X 67.4326,Y -120.8727,Z 188,A -54.6633,B 2.222,C 0.2603,E1 2.3181,E2 507.8615} C_DIS
LIN {X 63.5926,Y -122.9361,Z 188,A -56.2902,B 2.2219,C 0.2617,E1 2.3141,E2 509.4657} C_DIS
LIN {X 60.4494,Y -124.5119,Z 188,A -57.6998,B 2.2217,C 0.2634,E1 2.3106,E2 510.87} C_DIS
LIN {X 57.5473,Y -125.878,Z 188,A -58.9969,B 2.2215,C 0.265,E1 2.3073,E2 512.1638} C_DIS
LIN {X 54.1346,Y -127.3845,Z 188,A -60.4857,B 2.2213,C 0.2667,E1 2.3035,E2 513.6462} C_DIS
LIN {X 50.948,Y -128.6921,Z 188,A -61.8716,B 2.2211,C 0.2681,E1 2.2999,E2 515.0276} C_DIS
LIN {X 48.2536,Y -129.724,Z 188,A -63.0289,B 2.221,C 0.2693,E1 2.2969,E2 516.1806} C_DIS
LIN {X 45.0421,Y -130.8738,Z 188,A -64.4089,B 2.2208,C 0.2707,E1 2.2932,E2 517.5572} C_DIS
LIN {X 41.3116,Y -132.1011,Z 188,A -65.9951,B 2.2206,C 0.2721,E1 2.289,E2 519.1391} C_DIS
LIN {X 38.4579,Y -132.958,Z 188,A -67.1885,B 2.2205,C 0.2731,E1 2.2858,E2 520.3278} C_DIS
LIN {X 35.3666,Y -133.8131,Z 188,A -68.498,B 2.2204,C 0.2742,E1 2.2823,E2 521.6356} C_DIS
LIN {X 32.1381,Y -134.625,Z 188,A -69.8474,B 2.2202,C 0.2752,E1 2.2786,E2 522.982} C_DIS
LIN {X 28.4031,Y -135.4645,Z 188,A -71.4023,B 2.2201,C 0.2763,E1 2.2744,E2 524.5338} C_DIS
LIN {X 25.6943,Y -136.0021,Z 188,A -72.5449,B 2.22,C 0.2771,E1 2.2712,E2 525.6769} C_DIS
LIN {X 21.9775,Y -136.6541,Z 188,A -74.0607,B 2.2199,C 0.2779,E1 2.2671,E2 527.1874} C_DIS
LIN {X 18.7816,Y -137.1299,Z 188,A -75.378,B 2.2199,C 0.2786,E1 2.2634,E2 528.5027} C_DIS
LIN {X 15.8427,Y -137.4992,Z 188,A -76.5984,B 2.2197,C 0.2792,E1 2.26,E2 529.7229} C_DIS
LIN {X 12.4368,Y -137.8502,Z 188,A -77.9864,B 2.2197,C 0.2798,E1 2.2562,E2 531.1077} C_DIS
LIN {X 9.4206,Y -138.0885,Z 188,A -79.1917,B 2.2197,C 0.28,E1 2.2528,E2 532.3072} C_DIS
LIN {X 5.2405,Y -138.3088,Z 188,A -80.9578,B 2.2195,C 0.2808,E1 2.2479,E2 534.0787} C_DIS
LIN {X 2.0199,Y -138.3935,Z 188,A -82.2633,B 2.2195,C 0.281,E1 2.2442,E2 535.381} C_DIS
LIN {X 2.0199,Y -138.3935,Z 188,A -82.2633,B 2.2195,C 0.281,E1 2.2442,E2 535.381} C_DIS
Enddeposition()
LIN {X 1.0259,Y -139.2998,Z 188,A -82.2106,B 2.1908,C 0.2784,E1 2.2155,E2 535.302} C_DIS
Startdeposition()
$VEL.CP = VEL_PRINT
LIN {X 4.4141,Y -139.2384,Z 188,A -80.5338,B 2.191,C 0.2764,E1 2.2204,E2 533.5852} C_DIS
LIN {X 8.3882,Y -139.0545,Z 188,A -79.0419,B 2.191,C 0.2767,E1 2.2245,E2 532.1126} C_DIS
LIN {X 11.697,Y -138.8152,Z 188,A -77.6043,B 2.1911,C 0.2756,E1 2.2285,E2 530.664} C_DIS
LIN {X 15.7335,Y -138.4179,Z 188,A -75.842,B 2.1913,C 0.2742,E1 2.2335,E2 528.8877} C_DIS
LIN {X 19.3437,Y -137.958,Z 188,A -74.4879,B 2.1913,C 0.2742,E1 2.2372,E2 527.5527} C_DIS
LIN {X 23.007,Y -137.3941,Z 188,A -73.0915,B 2.1913,C 0.274,E1 2.241,E2 526.1732} C_DIS
LIN {X 29.5157,Y -136.1443,Z 188,A -70.4234,B 2.1915,C 0.2723,E1 2.2483,E2 523.5116} C_DIS
LIN {X 32.85,Y -135.3785,Z 188,A -68.9125,B 2.1918,C 0.2704,E1 2.2524,E2 521.9854} C_DIS
LIN {X 37.4534,Y -134.1777,Z 188,A -67.0997,B 2.1918,C 0.2695,E1 2.2573,E2 520.1914} C_DIS
LIN {X 40.3525,Y -133.3352,Z 188,A -65.9821,B 2.1919,C 0.2691,E1 2.2602,E2 519.0902} C_DIS
LIN {X 43.6248,Y -132.3005,Z 188,A -64.571,B 2.1921,C 0.2676,E1 2.264,E2 517.6783} C_DIS
LIN {X 46.9686,Y -131.1504,Z 188,A -63.018,B 2.1924,C 0.2654,E1 2.2682,E2 516.1106} C_DIS
LIN {X 50.2755,Y -129.9184,Z 188,A -61.8453,B 2.1924,C 0.2655,E1 2.2711,E2 514.9756} C_DIS
LIN {X 52.9653,Y -128.8474,Z 188,A -60.3495,B 2.1928,C 0.262,E1 2.2751,E2 513.4368} C_DIS
LIN {X 56.3757,Y -127.3909,Z 188,A -58.6047,B 2.1932,C 0.2585,E1 2.2797,E2 511.6603} C_DIS
LIN {X 59.848,Y -125.796,Z 188,A -57.5606,B 2.193,C 0.26,E1 2.2821,E2 510.6884} C_DIS
LIN {X 63.0784,Y -124.2074,Z 188,A -56.1062,B 2.1933,C 0.2581,E1 2.2858,E2 509.2366} C_DIS
LIN {X 66.1858,Y -122.5824,Z 188,A -54.6328,B 2.1935,C 0.2557,E1 2.2894,E2 507.7579} C_DIS
LIN {X 70.2717,Y -120.2868,Z 188,A -52.6445,B 2.1939,C 0.2523,E1 2.2943,E2 505.7598} C_DIS
LIN {X 74.2451,Y -117.8754,Z 188,A -50.8298,B 2.1942,C 0.2499,E1 2.2986,E2 503.9571} C_DIS
LIN {X 77.9146,Y -115.4828,Z 188,A -49.1197,B 2.1945,C 0.2475,E1 2.3025,E2 502.2583} C_DIS
LIN {X 81.3979,Y -113.0552,Z 188,A -47.3879,B 2.1948,C 0.2445,E1 2.3065,E2 500.5273} C_DIS
LIN {X 85.0124,Y -110.3629,Z 188,A -45.6169,B 2.1951,C 0.2417,E1 2.3104,E2 498.7662} C_DIS
LIN {X 88.5733,Y -107.5259,Z 188,A -43.8136,B 2.1954,C 0.2387,E1 2.3143,E2 496.9711} C_DIS
LIN {X 92.1344,Y -104.4901,Z 188,A -41.9905,B 2.1958,C 0.2357,E1 2.3181,E2 495.1604} C_DIS
LIN {X 95.6033,Y -101.3259,Z 188,A -40.1691,B 2.1961,C 0.2326,E1 2.3218,E2 493.3527} C_DIS
LIN {X 98.8845,Y -98.1263,Z 188,A -38.3628,B 2.1965,C 0.2293,E1 2.3254,E2 491.5557} C_DIS
LIN {X 102.0986,Y -94.7779,Z 188,A -36.5901,B 2.1968,C 0.2262,E1 2.3287,E2 489.8001} C_DIS
LIN {X 104.8747,Y -91.6965,Z 188,A -34.9078,B 2.1971,C 0.2227,E1 2.3319,E2 488.1198} C_DIS
LIN {X 107.8479,Y -88.1801,Z 188,A -33.1298,B 2.1975,C 0.2193,E1 2.335,E2 486.3562} C_DIS
LIN {X 110.5606,Y -84.7543,Z 188,A -31.394,B 2.1978,C 0.2157,E1 2.338,E2 484.6273} C_DIS
LIN {X 113.2359,Y -81.1453,Z 188,A -29.675,B 2.1981,C 0.2124,E1 2.3408,E2 482.9245} C_DIS
LIN {X 115.6896,Y -77.6075,Z 188,A -27.9549,B 2.1985,C 0.2085,E1 2.3435,E2 481.2098} C_DIS
LIN {X 117.6871,Y -74.5433,Z 188,A -26.1402,B 2.1991,C 0.2024,E1 2.3463,E2 479.3517} C_DIS
LIN {X 120.0889,Y -70.6086,Z 188,A -24.7781,B 2.1991,C 0.202,E1 2.3481,E2 478.061} C_DIS
LIN {X 122.1835,Y -66.9191,Z 188,A -23.1499,B 2.1994,C 0.1986,E1 2.3503,E2 476.4472} C_DIS
LIN {X 124.0943,Y -63.3006,Z 188,A -21.6127,B 2.1997,C 0.1955,E1 2.3523,E2 474.9283} C_DIS
LIN {X 126.5762,Y -58.1801,Z 188,A -19.2783,B 2.2002,C 0.1895,E1 2.3551,E2 472.593} C_DIS
LIN {X 128.3127,Y -54.2456,Z 188,A -17.6919,B 2.2005,C 0.1863,E1 2.3568,E2 471.03} C_DIS
LIN {X 129.7233,Y -50.7775,Z 188,A -16.2915,B 2.2008,C 0.1834,E1 2.3582,E2 469.6472} C_DIS
LIN {X 130.974,Y -47.4579,Z 188,A -15.1046,B 2.2008,C 0.1817,E1 2.3594,E2 468.4957} C_DIS
LIN {X 132.0615,Y -44.3427,Z 188,A -13.7541,B 2.2012,C 0.1782,E1 2.3606,E2 467.1451} C_DIS
LIN {X 132.9739,Y -41.5328,Z 188,A -12.3445,B 2.2016,C 0.1733,E1 2.3618,E2 465.7087} C_DIS
LIN {X 134.1581,Y -37.5235,Z 188,A -10.8192,B 2.2018,C 0.1702,E1 2.363,E2 464.208} C_DIS
LIN {X 135.2605,Y -33.3382,Z 188,A -8.2562,B 2.2027,C 0.1589,E1 2.3647,E2 461.5384} C_DIS
LIN {X 136.7764,Y -26.4338,Z 188,A -6.4196,B 2.2026,C 0.1597,E1 2.3657,E2 459.8437} C_DIS
LIN {X 137.3722,Y -23.1383,Z 188,A -4.8645,B 2.203,C 0.1544,E1 2.3664,E2 458.264} C_DIS
LIN {X 137.8863,Y -19.8459,Z 188,A -3.9201,B 2.203,C 0.1541,E1 2.3668,E2 457.3753} C_DIS
LIN {X 138.2959,Y -16.7569,Z 188,A -2.6593,B 2.2032,C 0.1507,E1 2.3672,E2 456.1164} C_DIS
LIN {X 138.678,Y -13.2251,Z 188,A -1.2132,B 2.2035,C 0.1467,E1 2.3676,E2 454.6714} C_DIS
LIN {X 139.03,Y -8.7874,Z 188,A 0.4166,B 2.2037,C 0.1432,E1 2.3679,E2 453.067} C_DIS
LIN {X 139.2079,Y -5.2638,Z 188,A 1.8279,B 2.204,C 0.1395,E1 2.3681,E2 451.6601} C_DIS
LIN {X 139.3054,Y -0.8729,Z 188,A 3.5166,B 2.2042,C 0.1354,E1 2.3681,E2 449.9857} C_DIS
LIN {X 139.2721,Y 3.1992,Z 188,A 5.1578,B 2.2045,C 0.131,E1 2.3681,E2 448.348} C_DIS
LIN {X 139.1265,Y 7.0946,Z 188,A 6.6029,B 2.2047,C 0.1277,E1 2.3679,E2 446.9227} C_DIS
LIN {X 138.8698,Y 11.0504,Z 188,A 8.23,B 2.2049,C 0.1232,E1 2.3676,E2 445.2951} C_DIS
LIN {X 138.5149,Y 14.8355,Z 188,A 9.4956,B 2.205,C 0.1213,E1 2.3673,E2 444.0675} C_DIS
LIN {X 138.1528,Y 17.8974,Z 188,A 10.7457,B 2.2052,C 0.1179,E1 2.3668,E2 442.8191} C_DIS
LIN {X 137.7,Y 21.0999,Z 188,A 12.7365,B 2.2057,C 0.1088,E1 2.366,E2 440.741} C_DIS
LIN {X 136.6786,Y 26.9451,Z 188,A 14.5621,B 2.2057,C 0.1071,E1 2.365,E2 438.9949} C_DIS
LIN {X 135.6212,Y 31.8425,Z 188,A 16.397,B 2.206,C 0.1032,E1 2.3639,E2 437.1884} C_DIS
LIN {X 134.6961,Y 35.5459,Z 188,A 17.9328,B 2.2062,C 0.0992,E1 2.3628,E2 435.6562} C_DIS
LIN {X 133.3503,Y 40.303,Z 188,A 19.6829,B 2.2062,C 0.096,E1 2.3615,E2 433.9419} C_DIS
LIN {X 132.2458,Y 43.7893,Z 188,A 21.1119,B 2.2064,C 0.0925,E1 2.3603,E2 432.5219} C_DIS
LIN {X 131.1272,Y 47.033,Z 188,A 22.3173,B 2.2065,C 0.0904,E1 2.3592,E2 431.3424} C_DIS
LIN {X 129.8824,Y 50.3682,Z 188,A 23.7623,B 2.2067,C 0.0867,E1 2.3578,E2 429.8992} C_DIS
LIN {X 128.6577,Y 53.4194,Z 188,A 25.0823,B 2.2068,C 0.0834,E1 2.3564,E2 428.5828} C_DIS
LIN {X 127.286,Y 56.6103,Z 188,A 26.3941,B 2.2069,C 0.0806,E1 2.3549,E2 427.2854} C_DIS
LIN {X 126.0645,Y 59.2859,Z 188,A 27.5762,B 2.207,C 0.0777,E1 2.3535,E2 426.1065} C_DIS
LIN {X 124.2617,Y 62.9718,Z 188,A 29.1654,B 2.2071,C 0.0741,E1 2.3516,E2 424.5292} C_DIS
LIN {X 122.4635,Y 66.4059,Z 188,A 30.7807,B 2.2073,C 0.07,E1 2.3494,E2 422.9108} C_DIS
LIN {X 120.2014,Y 70.4171,Z 188,A 32.5541,B 2.2073,C 0.0662,E1 2.347,E2 421.1522} C_DIS
LIN {X 117.7508,Y 74.4424,Z 188,A 34.5081,B 2.2075,C 0.0614,E1 2.3441,E2 419.1957} C_DIS
LIN {X 114.8895,Y 78.7865,Z 188,A 36.4455,B 2.2076,C 0.0578,E1 2.3411,E2 417.2834} C_DIS
LIN {X 112.0641,Y 82.7566,Z 188,A 38.3111,B 2.2077,C 0.0542,E1 2.3381,E2 415.4349} C_DIS
LIN {X 105.9116,Y 90.4974,Z 188,A 42.0166,B 2.2079,C 0.0477,E1 2.3317,E2 411.7744} C_DIS
LIN {X 103.3333,Y 93.4302,Z 188,A 43.7296,B 2.2079,C 0.0434,E1 2.3284,E2 410.0478} C_DIS
LIN {X 100.1561,Y 96.8281,Z 188,A 45.5327,B 2.208,C 0.0401,E1 2.325,E2 408.2581} C_DIS
LIN {X 96.8917,Y 100.0945,Z 188,A 47.1215,B 2.208,C 0.0384,E1 2.3219,E2 406.7081} C_DIS
LIN {X 91.2799,Y 105.238,Z 188,A 50.2475,B 2.2081,C 0.0323,E1 2.3155,E2 403.5826} C_DIS
LIN {X 87.9887,Y 108.0044,Z 188,A 52.0413,B 2.2081,C 0.0287,E1 2.3116,E2 401.7855} C_DIS
LIN {X 84.5324,Y 110.7303,Z 188,A 53.7733,B 2.2082,C 0.026,E1 2.3078,E2 400.0633} C_DIS
LIN {X 81.4318,Y 113.0307,Z 188,A 55.3645,B 2.2082,C 0.0231,E1 2.3042,E2 398.4716} C_DIS
LIN {X 77.5008,Y 115.7609,Z 188,A 57.2198,B 2.2082,C 0.0205,E1 2.2999,E2 396.6304} C_DIS
LIN {X 73.4667,Y 118.3621,Z 188,A 59.0852,B 2.2083,C 0.018,E1 2.2955,E2 394.7786} C_DIS
LIN {X 69.4835,Y 120.7439,Z 188,A 60.9587,B 2.2083,C 0.0153,E1 2.291,E2 392.9096} C_DIS
LIN {X 65.5048,Y 122.9478,Z 188,A 62.7967,B 2.2083,C 0.0128,E1 2.2865,E2 391.0758} C_DIS
LIN {X 61.7819,Y 124.8574,Z 188,A 64.2728,B 2.2083,C 0.0119,E1 2.2829,E2 389.63} C_DIS
LIN {X 58.7907,Y 126.2939,Z 188,A 65.6784,B 2.2083,C 0.0098,E1 2.2793,E2 388.2196} C_DIS
LIN {X 55.5358,Y 127.7584,Z 188,A 67.0784,B 2.2083,C 0.0083,E1 2.2758,E2 386.8282} C_DIS
LIN {X 52.3064,Y 129.1142,Z 188,A 68.492,B 2.2083,C 0.0067,E1 2.2721,E2 385.4181} C_DIS
LIN {X 49.1943,Y 130.332,Z 188,A 69.7038,B 2.2083,C 0.0061,E1 2.269,E2 384.2266} C_DIS
LIN {X 46.0219,Y 131.4859,Z 188,A 71.2321,B 2.2083,C 0.0037,E1 2.2649,E2 382.6813} C_DIS
LIN {X 41.611,Y 132.9496,Z 188,A 73.4862,B 2.2083,C -0.0002,E1 2.2588,E2 380.3856} C_DIS
LIN {X 37.6947,Y 134.1102,Z 188,A 74.6609,B 2.2083,C 0.0011,E1 2.2558,E2 379.2733} C_DIS
LIN {X 34.4533,Y 134.9793,Z 188,A 76.0286,B 2.2083,C 0,E1 2.2521,E2 377.9075} C_DIS
LIN {X 30.7509,Y 135.8708,Z 188,A 78.1124,B 2.2083,C -0.0042,E1 2.2463,E2 375.7606} C_DIS
LIN {X 26.128,Y 136.8348,Z 188,A 79.3166,B 2.2083,C -0.0015,E1 2.2432,E2 374.6475} C_DIS
LIN {X 21.2537,Y 137.6762,Z 188,A 81.4773,B 2.2083,C -0.0035,E1 2.2372,E2 372.472} C_DIS
LIN {X 17.7737,Y 138.169,Z 188,A 82.9842,B 2.2083,C -0.0046,E1 2.233,E2 370.9582} C_DIS
LIN {X 13.8728,Y 138.6158,Z 188,A 84.5683,B 2.2083,C -0.0052,E1 2.2286,E2 369.3785} C_DIS
LIN {X 9.8936,Y 138.9556,Z 188,A 86.1739,B 2.2083,C -0.0057,E1 2.2241,E2 367.778} C_DIS
LIN {X 5.7214,Y 139.19,Z 188,A 87.8699,B 2.2083,C -0.0062,E1 2.2194,E2 366.0853} C_DIS
LIN {X 2.0549,Y 139.2924,Z 188,A 89.4448,B 2.2083,C -0.0069,E1 2.215,E2 364.5029} C_DIS
LIN {X -2.2454,Y 139.2892,Z 188,A 91.2001,B 2.2083,C -0.0071,E1 2.2101,E2 362.75} C_DIS
LIN {X -6.5055,Y 139.1561,Z 188,A 92.8853,B 2.2083,C -0.0069,E1 2.2054,E2 361.0739} C_DIS
LIN {X -10.0868,Y 138.9415,Z 188,A 94.3319,B 2.2083,C -0.0067,E1 2.2013,E2 359.6314} C_DIS
LIN {X -13.9149,Y 138.6118,Z 188,A 96.0313,B 2.2083,C -0.0072,E1 2.1966,E2 357.9184} C_DIS
LIN {X -17.952,Y 138.1456,Z 188,A 97.3673,B 2.2083,C -0.0054,E1 2.193,E2 356.6238} C_DIS
LIN {X -25.9845,Y 136.8622,Z 188,A 100.7074,B 2.2083,C -0.0045,E1 2.1838,E2 353.2864} C_DIS
LIN {X -31.8182,Y 135.627,Z 188,A 103.5527,B 2.2083,C -0.0051,E1 2.1758,E2 350.3949} C_DIS
LIN {X -35.151,Y 134.8014,Z 188,A 105.0122,B 2.2083,C -0.0046,E1 2.1719,E2 348.9303} C_DIS
LIN {X -38.6443,Y 133.8405,Z 188,A 106.4013,B 2.2083,C -0.0033,E1 2.1682,E2 347.5544} C_DIS
LIN {X -42.1052,Y 132.7917,Z 188,A 107.9298,B 2.2083,C -0.0025,E1 2.1641,E2 346.0217} C_DIS
LIN {X -45.5868,Y 131.6367,Z 188,A 109.3668,B 2.2083,C -0.0011,E1 2.1603,E2 344.5943} C_DIS
LIN {X -48.6439,Y 130.5381,Z 188,A 110.8191,B 2.2083,C -0.0005,E1 2.1564,E2 343.1287} C_DIS
LIN {X -52.5686,Y 129.0085,Z 188,A 112.9901,B 2.2083,C -0.0005,E1 2.1507,E2 340.905} C_DIS
LIN {X -56.3233,Y 127.4143,Z 188,A 114.3635,B 2.2083,C 0.0022,E1 2.1472,E2 339.57} C_DIS
LIN {X -59.5712,Y 125.9282,Z 188,A 115.9762,B 2.2083,C 0.0032,E1 2.1431,E2 337.9405} C_DIS
LIN {X -64.2861,Y 123.5878,Z 188,A 118.0569,B 2.2083,C 0.0059,E1 2.1379,E2 335.8715} C_DIS
LIN {X -68.0776,Y 121.5418,Z 188,A 120.1105,B 2.2083,C 0.0071,E1 2.1328,E2 333.7846} C_DIS
LIN {X -70.928,Y 119.901,Z 188,A 122.0017,B 2.2083,C 0.0071,E1 2.1281,E2 331.8277} C_DIS
LIN {X -75.9181,Y 116.8048,Z 188,A 123.7942,B 2.2083,C 0.0124,E1 2.1241,E2 330.1138} C_DIS
LIN {X -82.5881,Y 112.1879,Z 188,A 127.2228,B 2.2083,C 0.0171,E1 2.1162,E2 326.6762} C_DIS
LIN {X -86.1594,Y 109.4691,Z 188,A 129.1681,B 2.2083,C 0.0198,E1 2.1119,E2 324.72} C_DIS
LIN {X -89.7623,Y 106.5351,Z 188,A 131.1814,B 2.2083,C 0.0227,E1 2.1075,E2 322.6954} C_DIS
LIN {X -93.1078,Y 103.6238,Z 188,A 133.0835,B 2.2083,C 0.0257,E1 2.1035,E2 320.785} C_DIS
LIN {X -96.5798,Y 100.3965,Z 188,A 135.1334,B 2.2082,C 0.029,E1 2.0994,E2 318.724} C_DIS
LIN {X -99.7919,Y 97.2043,Z 188,A 137.073,B 2.2082,C 0.0323,E1 2.0955,E2 316.7762} C_DIS
LIN {X -102.8208,Y 93.9944,Z 188,A 138.982,B 2.2081,C 0.0356,E1 2.0919,E2 314.8568} C_DIS
LIN {X -105.7989,Y 90.6292,Z 188,A 140.8729,B 2.2081,C 0.0393,E1 2.0884,E2 312.9619} C_DIS
LIN {X -108.6631,Y 87.1744,Z 188,A 142.8448,B 2.208,C 0.0429,E1 2.0849,E2 310.9757} C_DIS
LIN {X -113.808,Y 80.3409,Z 188,A 146.5255,B 2.2078,C 0.0502,E1 2.0788,E2 307.2773} C_DIS
LIN {X -116.3047,Y 76.6821,Z 188,A 148.4591,B 2.2078,C 0.0541,E1 2.0757,E2 305.3311} C_DIS
LIN {X -118.7276,Y 72.8745,Z 188,A 150.1884,B 2.2076,C 0.0587,E1 2.0732,E2 303.619} C_DIS
LIN {X -120.8098,Y 69.369,Z 188,A 152.237,B 2.2076,C 0.0619,E1 2.0702,E2 301.5251} C_DIS
LIN {X -122.9997,Y 65.4059,Z 188,A 154.1784,B 2.2074,C 0.0662,E1 2.0676,E2 299.5751} C_DIS
LIN {X -124.7937,Y 61.9111,Z 188,A 155.9523,B 2.2073,C 0.0699,E1 2.0654,E2 297.7822} C_DIS
LIN {X -126.7724,Y 57.7557,Z 188,A 157.7286,B 2.2071,C 0.0749,E1 2.0633,E2 296.0221} C_DIS
LIN {X -130.2281,Y 49.4716,Z 188,A 162.2088,B 2.2068,C 0.0829,E1 2.0585,E2 291.4446} C_DIS
LIN {X -131.6178,Y 45.6413,Z 188,A 163.4526,B 2.2066,C 0.0881,E1 2.0574,E2 290.2571} C_DIS
LIN {X -132.6456,Y 42.5625,Z 188,A 164.8272,B 2.2065,C 0.0916,E1 2.0562,E2 288.8784} C_DIS
LIN {X -133.5971,Y 39.4758,Z 188,A 166.376,B 2.2063,C 0.0947,E1 2.0549,E2 287.3025} C_DIS
LIN {X -134.3607,Y 36.7989,Z 188,A 167.9434,B 2.2063,C 0.097,E1 2.0537,E2 285.6818} C_DIS
LIN {X -135.2644,Y 33.3233,Z 188,A 169.2957,B 2.2061,C 0.1012,E1 2.0528,E2 284.3465} C_DIS
LIN {X -136.0453,Y 29.9744,Z 188,A 170.6213,B 2.2059,C 0.1053,E1 2.052,E2 283.0333} C_DIS
LIN {X -136.7798,Y 26.4158,Z 188,A 172.3078,B 2.2057,C 0.109,E1 2.0511,E2 281.3231} C_DIS
LIN {X -137.4265,Y 22.8128,Z 188,A 174.0314,B 2.2055,C 0.1128,E1 2.0503,E2 279.5725} C_DIS
LIN {X -138.2191,Y 17.3913,Z 188,A 176.6666,B 2.2052,C 0.1183,E1 2.0493,E2 276.8893} C_DIS
LIN {X -138.6256,Y 13.7703,Z 188,A 177.8793,B 2.2049,C 0.1231,E1 2.0489,E2 275.7147} C_DIS
LIN {X -138.9338,Y 10.1927,Z 188,A 179.3734,B 2.2047,C 0.1272,E1 2.0486,E2 274.2193} C_DIS
LIN {X -139.2173,Y 5.0208,Z 188,A -178.0435,B 2.2044,C 0.1323,E1 2.0483,E2 271.5787} C_DIS
LIN {X -139.3059,Y -0.8058,Z 188,A -175.6068,B 2.204,C 0.1389,E1 2.0483,E2 269.1383} C_DIS
LIN {X -139.2236,Y -4.8595,Z 188,A -173.4465,B 2.2038,C 0.1427,E1 2.0484,E2 266.9144} C_DIS
LIN {X -139.021,Y -8.9324,Z 188,A -171.8639,B 2.2034,C 0.1476,E1 2.0487,E2 265.3453} C_DIS
LIN {X -138.6079,Y -13.9549,Z 188,A -169.901,B 2.203,C 0.1536,E1 2.0492,E2 263.398} C_DIS
LIN {X -138.1768,Y -17.7139,Z 188,A -168.1872,B 2.2028,C 0.1576,E1 2.0498,E2 261.6643} C_DIS
LIN {X -137.5963,Y -21.7697,Z 188,A -166.3008,B 2.2024,C 0.1618,E1 2.0506,E2 259.7523} C_DIS
LIN {X -136.9061,Y -25.7554,Z 188,A -164.6195,B 2.2021,C 0.1664,E1 2.0514,E2 258.0696} C_DIS
LIN {X -136.1938,Y -29.2863,Z 188,A -163.0861,B 2.2018,C 0.1703,E1 2.0523,E2 256.53} C_DIS
LIN {X -135.4981,Y -32.354,Z 188,A -161.7098,B 2.2015,C 0.1737,E1 2.0532,E2 255.1435} C_DIS
LIN {X -134.6552,Y -35.699,Z 188,A -160.1937,B 2.2013,C 0.1773,E1 2.0542,E2 253.6151} C_DIS
LIN {X -133.781,Y -38.8475,Z 188,A -158.7311,B 2.201,C 0.1807,E1 2.0554,E2 252.1373} C_DIS
LIN {X -132.8485,Y -41.9275,Z 188,A -157.3283,B 2.2007,C 0.184,E1 2.0565,E2 250.7246} C_DIS
LIN {X -131.7194,Y -45.3483,Z 188,A -155.9889,B 2.2003,C 0.1882,E1 2.0577,E2 249.4049} C_DIS
LIN {X -129.9966,Y -50.0745,Z 188,A -153.5605,B 2.2,C 0.1928,E1 2.0601,E2 246.9294} C_DIS
LIN {X -128.6676,Y -53.3959,Z 188,A -151.8352,B 2.1997,C 0.196,E1 2.062,E2 245.1707} C_DIS
LIN {X -126.6499,Y -58.0206,Z 188,A -149.7601,B 2.1992,C 0.2012,E1 2.0643,E2 243.0965} C_DIS
LIN {X -125.0575,Y -61.3762,Z 188,A -148.2871,B 2.1988,C 0.2051,E1 2.0661,E2 241.6313} C_DIS
LIN {X -123.6556,Y -64.1569,Z 188,A -146.7492,B 2.1986,C 0.2076,E1 2.0681,E2 240.0594} C_DIS
LIN {X -121.5723,Y -68.0233,Z 188,A -144.7809,B 2.1982,C 0.2115,E1 2.0708,E2 238.0698} C_DIS
LIN {X -119.2907,Y -71.9491,Z 188,A -142.8753,B 2.1978,C 0.2158,E1 2.0735,E2 236.1596} C_DIS
LIN {X -117.1368,Y -75.4057,Z 188,A -141.042,B 2.1975,C 0.2193,E1 2.0763,E2 234.3054} C_DIS
LIN {X -114.5886,Y -79.2246,Z 188,A -139.0395,B 2.1971,C 0.2232,E1 2.0795,E2 232.2879} C_DIS
LIN {X -110.5494,Y -84.769,Z 188,A -136.1638,B 2.1965,C 0.2291,E1 2.0843,E2 229.4054} C_DIS
LIN {X -107.8423,Y -88.187,Z 188,A -134.2256,B 2.1961,C 0.2325,E1 2.0877,E2 227.4478} C_DIS
LIN {X -104.8811,Y -91.689,Z 188,A -132.5056,B 2.1957,C 0.2368,E1 2.0908,E2 225.7509} C_DIS
LIN {X -102.5768,Y -94.2599,Z 188,A -130.7558,B 2.1955,C 0.2386,E1 2.0941,E2 223.9563} C_DIS
LIN {X -98.9555,Y -98.0549,Z 188,A -128.1138,B 2.1952,C 0.2411,E1 2.0994,E2 221.248} C_DIS
LIN {X -95.8831,Y -101.0619,Z 188,A -126.6169,B 2.1947,C 0.2452,E1 2.1024,E2 219.7886} C_DIS
LIN {X -92.5141,Y -104.1545,Z 188,A -124.8444,B 2.1943,C 0.2488,E1 2.106,E2 218.0312} C_DIS
LIN {X -89.5729,Y -106.694,Z 188,A -123.0575,B 2.1941,C 0.2509,E1 2.1099,E2 216.2184} C_DIS
LIN {X -86.1743,Y -109.4575,Z 188,A -121.1545,B 2.1938,C 0.2534,E1 2.1141,E2 214.3015} C_DIS
LIN {X -82.2555,Y -112.4323,Z 188,A -119.0694,B 2.1935,C 0.2563,E1 2.1188,E2 212.2079} C_DIS
LIN {X -78.4976,Y -115.0878,Z 188,A -117.0816,B 2.1932,C 0.2587,E1 2.1234,E2 210.2069} C_DIS
LIN {X -74.6794,Y -117.6013,Z 188,A -115.126,B 2.1929,C 0.2609,E1 2.128,E2 208.2408} C_DIS
LIN {X -70.8503,Y -119.947,Z 188,A -113.2768,B 2.1926,C 0.2633,E1 2.1324,E2 206.3911} C_DIS
LIN {X -67.0585,Y -122.1075,Z 188,A -111.3761,B 2.1924,C 0.265,E1 2.1371,E2 204.4756} C_DIS
LIN {X -63.413,Y -124.0371,Z 188,A -109.8848,B 2.1921,C 0.2677,E1 2.1407,E2 203.0123} C_DIS
LIN {X -60.4302,Y -125.5178,Z 188,A -108.3303,B 2.1921,C 0.2684,E1 2.1447,E2 201.4321} C_DIS
LIN {X -57.1717,Y -127.0349,Z 188,A -106.8645,B 2.1918,C 0.2698,E1 2.1484,E2 199.9677} C_DIS
LIN {X -53.9859,Y -128.4211,Z 188,A -105.3788,B 2.1918,C 0.2709,E1 2.1523,E2 198.4739} C_DIS
LIN {X -50.741,Y -129.7375,Z 188,A -103.9328,B 2.1916,C 0.2721,E1 2.156,E2 197.0269} C_DIS
LIN {X -47.497,Y -130.9599,Z 188,A -102.4613,B 2.1915,C 0.273,E1 2.1599,E2 195.5486} C_DIS
LIN {X -43.1081,Y -132.4711,Z 188,A -100.2807,B 2.1915,C 0.273,E1 2.1658,E2 193.3298} C_DIS
LIN {X -37.8335,Y -134.0714,Z 188,A -98.2345,B 2.1911,C 0.2754,E1 2.1712,E2 191.3137} C_DIS
LIN {X -33.6721,Y -135.1776,Z 188,A -96.1967,B 2.1912,C 0.275,E1 2.1769,E2 189.2382} C_DIS
LIN {X -28.4198,Y -136.3788,Z 188,A -94.1144,B 2.191,C 0.2765,E1 2.1825,E2 187.1738} C_DIS
LIN {X -24.3087,Y -137.1699,Z 188,A -92.4189,B 2.191,C 0.2771,E1 2.1872,E2 185.4814} C_DIS
LIN {X -19.8791,Y -137.8815,Z 188,A -90.6109,B 2.1909,C 0.2777,E1 2.1922,E2 183.6778} C_DIS
LIN {X -16.8476,Y -138.285,Z 188,A -89.4902,B 2.1907,C 0.2786,E1 2.1952,E2 182.5758} C_DIS
LIN {X -13.4579,Y -138.6556,Z 188,A -87.929,B 2.1908,C 0.2778,E1 2.1996,E2 180.9918} C_DIS
LIN {X -9.5623,Y -138.9798,Z 188,A -86.2513,B 2.1908,C 0.2774,E1 2.2043,E2 179.3037} C_DIS
LIN {X -5.5068,Y -139.1984,Z 188,A -84.7321,B 2.1908,C 0.2781,E1 2.2085,E2 177.8048} C_DIS
LIN {X -2.1768,Y -139.2903,Z 188,A -83.2713,B 2.1908,C 0.2774,E1 2.2127,E2 176.3307} C_DIS
LIN {X 1.0259,Y -139.2998,Z 188,A -82.2079,B 2.1908,C 0.2785,E1 2.2156,E2 175.3019} C_DIS
Enddeposition()
LIN {X 1.0259,Y -139.2998,Z 188,A -82.2079,B 2.1908,C 0.2785,E1 2.2156,E2 175.3019} C_DIS
Startdeposition()
$VEL.CP = VEL_PRINT
LIN {X -0.4109,Y -140.2065,Z 188,A -83.174,B 2.16,C 0.2805,E1 2.1822,E2 176.3593} C_DIS
LIN {X -4.2668,Y -140.1421,Z 188,A -84.8181,B 2.16,C 0.2811,E1 2.1776,E2 178.0136} C_DIS
LIN {X -8.5151,Y -139.9478,Z 188,A -86.4084,B 2.16,C 0.2805,E1 2.1732,E2 179.5841} C_DIS
LIN {X -11.8608,Y -139.7039,Z 188,A -87.8651,B 2.16,C 0.2809,E1 2.1691,E2 181.0533} C_DIS
LIN {X -16.3566,Y -139.2493,Z 188,A -89.694,B 2.16,C 0.2807,E1 2.164,E2 182.8805} C_DIS
LIN {X -19.9928,Y -138.7737,Z 188,A -91.1602,B 2.16,C 0.2803,E1 2.16,E2 184.3428} C_DIS
LIN {X -23.3438,Y -138.2496,Z 188,A -92.5621,B 2.16,C 0.28,E1 2.1561,E2 185.7474} C_DIS
LIN {X -26.6766,Y -137.6456,Z 188,A -93.9585,B 2.16,C 0.2797,E1 2.1523,E2 187.1461} C_DIS
LIN {X -29.979,Y -136.9643,Z 188,A -95.8333,B 2.1599,C 0.2816,E1 2.1469,E2 189.0902} C_DIS
LIN {X -34.311,Y -135.9433,Z 188,A -96.9246,B 2.1604,C 0.2773,E1 2.1443,E2 190.0811} C_DIS
LIN {X -37.05,Y -135.2243,Z 188,A -98.9152,B 2.16,C 0.2806,E1 2.1386,E2 192.1878} C_DIS
LIN {X -41.717,Y -133.858,Z 188,A -100.9139,B 2.1601,C 0.2794,E1 2.1332,E2 194.1886} C_DIS
LIN {X -46.152,Y -132.3926,Z 188,A -102.3012,B 2.1606,C 0.2757,E1 2.1297,E2 195.5042} C_DIS
LIN {X -49.4773,Y -131.1863,Z 188,A -103.7639,B 2.1607,C 0.2747,E1 2.1259,E2 196.9696} C_DIS
LIN {X -52.8354,Y -129.8706,Z 188,A -105.2357,B 2.1609,C 0.2735,E1 2.122,E2 198.4415} C_DIS
LIN {X -55.888,Y -128.5859,Z 188,A -106.6882,B 2.1609,C 0.2726,E1 2.1183,E2 199.908} C_DIS
LIN {X -59.2822,Y -127.0574,Z 188,A -108.2013,B 2.1612,C 0.2711,E1 2.1144,E2 201.4202} C_DIS
LIN {X -62.7719,Y -125.3718,Z 188,A -109.9795,B 2.1612,C 0.2703,E1 2.1099,E2 203.2256} C_DIS
LIN {X -66.718,Y -123.3173,Z 188,A -111.8158,B 2.1615,C 0.2683,E1 2.1053,E2 205.0646} C_DIS
LIN {X -70.6978,Y -121.0796,Z 188,A -113.7359,B 2.1618,C 0.2662,E1 2.1007,E2 206.9924} C_DIS
LIN {X -74.5118,Y -118.7705,Z 188,A -115.6349,B 2.1621,C 0.2641,E1 2.0961,E2 208.9021} C_DIS
LIN {X -78.3171,Y -116.2964,Z 188,A -117.5529,B 2.1623,C 0.2618,E1 2.0916,E2 210.829} C_DIS
LIN {X -82.1579,Y -113.6151,Z 188,A -119.6943,B 2.1626,C 0.2598,E1 2.0867,E2 213.0015} C_DIS
LIN {X -84.8459,Y -111.6227,Z 188,A -120.953,B 2.1629,C 0.2573,E1 2.0839,E2 214.2454} C_DIS
LIN {X -88.5363,Y -108.7183,Z 188,A -122.9313,B 2.1632,C 0.2544,E1 2.0795,E2 216.2318} C_DIS
LIN {X -93.1458,Y -104.7964,Z 188,A -125.2041,B 2.1638,C 0.2496,E1 2.0748,E2 218.4769} C_DIS
Enddeposition()
END
